ACTION aP15_FormTransporters:
(********Transporter przed dozownikami*************)
tofbFormTransportersDispencerSlow			(IN:=bFormTransportersDispencerSlowSpeedPulse, 	PT:=T#60S);
tonbFormTransportersDispencerResetSpeed		(IN:=bFormTransportersDispencerResetSpeed, 		PT:=T#5S);
tonQueBeforeScrewers						(IN:=P10_GripperScrewer.IbGripperScrewersSixthFormCheckFormSensor, PT:=T#1500mS);
tonQueAfterScrewers							(IN:=P11_CapCorrectCheck.IbCapCorrectCheckAfterScrewerFormSensor AND P11_CapCorrectCheck.IbCapCorrectCheckDialAfterScrewerFormSensor, PT:=T#2S);
tonQueAfterPlatin							(IN:=MAIN.IbLidSealerAfterSensor, PT:=T#3S);
tonQueBeforeDispencers						(IN:=MAIN.IbFormCheckFormSensor, PT:=T#2S);
tonDelayedStartAfterDisp					(IN:=NOT P09_CapPuttedCheck.fbIbCapPuttedCheckFormSensor.bOUT, PT:=T#1.5S);
IF GVL.bFormTransportersEnable AND (P00_PackML.fbPMLAuto.ePMLState = E_PMLState.ePMLState_EXECUTE)  THEN
	IF NOT VIS.bDosingTwoPhasesShow  THEN
		bFormTransportersDispencerCmdStart := TRUE;
	ELSIF VIS.bDosingTwoPhasesShow AND	NOT bFormTransportersScrewerStop AND NOT tonQueAfterPlatin.q THEN
		bFormTransportersDispencerCmdStart := TRUE;	
	END_IF
	bFormTransportersDispencerSlowSpeedPulse	:=	FALSE;
	(*Spowalnianie transportera*)	
	IF tofbFormTransportersDispencerSlow.Q AND NOT tonbFormTransportersDispencerResetSpeed.Q THEN
		bFormTransportersDispencerSlowSpeed	:= NOT VIS.bCapPuttedCheckIgnoreErrors; 
	ELSE
		bFormTransportersDispencerSlowSpeed	:= FALSE;
	END_IF
	IF bDosingTwoPhases THEN
		bFormTransportersDispencerSlowSpeed	:= TRUE;
	END_IF	
END_IF
	(*Wydmuch na tym transporterze*)
	QbBlowAfterGripperScrewer :=	bFormTransportersDispencerSlowSpeed;
(********Koniec Transporter przed dozownikami********)
	
(********Transporter za dozownikami*************)
tonbFormTransportersScrewerStop	(IN:=	(P05_Weight.eWeightStationRunningState = E_WeightLiftStationState.eStorageOfForms) AND 
										P05_Weight.fbWeightStation.iFormsCounterWeight1 >=3 AND 
										P05_Weight.fbWeightStation.iFormsCounterWeight2 >=3 AND 
										P05_Weight.fbWeightStation.iFormsCounterWeight3 >=3 AND 
										P05_Weight.fbWeightStation.iFormsCounterWeight4 >=3,
									PT:=T#500MS);
tofFormTransportersScrewerSlowSpeed	(IN:=P00_ReadRFIDCard.bReadedCardCapSorter AND bDosingTwoPhases, PT:=T#2S500MS);

IF 	P10_GripperScrewer.fbGripperScrewersDragStation.eRunningState = E_DragStationState.eEndingOfDrag  OR tonThirdFormCheckFormSensor.q THEN
//IF 	P10_GripperScrewer.fbGripperScrewersDragStation.eRunningState = E_DragStationState.eDraging AND P10_GripperScrewer.QbGripperScrewersDragLeadBefore1Actuator THEN
	bFormTransportersScrewerStop			:= FALSE;
END_IF


IF tonLongDelayAfterStart.Q AND
		eBeforeCapSorterPackageState[4].bFormPresent  AND
		(tonCapSorterFourthFormatSensorAnRegister.Q AND iCapSorterDragFormCounter >= 4)AND 
		MAIN.IbCapSorterBeforeFourthFormCheckFormSensor 
		THEN
			IF 
				NOT (
					(P05_Weight.eWeightStationRunningState = E_WeightLiftStationState.eStorageOfForms) AND 
					P05_Weight.fbWeightStation.iFormsCounterWeight1 =3 AND 
					P05_Weight.fbWeightStation.iFormsCounterWeight2 =3 AND 
					P05_Weight.fbWeightStation.iFormsCounterWeight3 =3 AND 
					P05_Weight.fbWeightStation.iFormsCounterWeight4 =3 
					)
				AND NOT bFormTransportersScrewerStop	
				//?AND NOT bLidFeederEnable
				(*AND NOT bDosingTwoPhases*)
				AND NOT bPhaseChanging
				AND tonDelayAfterStart.Q
				//AND (tonQueAfterScrewers.Q OR tonQueBeforeScrewers.Q)  //vs testy
			THEN
				bFormTransportersScrewerStop				:= 	TRUE;
			END_IF
		//bFormTransportersScrewerStop				:= 	TRUE;
END_IF
tonQueAfterScrewers.Q; tonQueBeforeScrewers.Q;
//IF bFormTransportersEnable AND (P00_PackML.fbPMLAuto.ePMLState = E_PMLState.ePMLState_EXECUTE)THEN //dp
IF bDelayAfterStart AND (*tonDelayAfterStart.Q AND*) bFormTransportersEnable AND (P00_PackML.fbPMLAuto.ePMLState = E_PMLState.ePMLState_EXECUTE OR 
		P00_PackML.fbPMLAuto.ePMLState = E_PMLState.ePMLState_STOPPING) (*AND tonDelayedStartAfterDisp.q co to*) THEN
	bFormTransportersScrewerCmdStart 			:= TRUE;
	tonbCapSorterOrCapSorterDragError.Q; 		//Spowalnianie transportera dla wag
	IF bFormTransportersScrewerStop	(*AND NOT tonbCapSorterOrCapSorterDragError.Q)*) THEN //Zatrzymywanie
		bFormTransportersScrewerCmdStart 		:= FALSE;
		
	END_IF
	//Vasyl na prośbę Karola
	(*IF (VIS.bDosingTwoPhasesShow OR vis.bLidFeederEnableShow) AND	tonQueAfterPlatin.Q OR bFormTransportersScrewerStop AND tonQueBeforeDispencers.q THEN
		bFormTransportersDispencerCmdStart 		:= FALSE;
	END_IF*)
END_IF

(********Transporter za sorterem nasadek*************)
IF bFormTransportersEnable AND (P00_PackML.fbPMLAuto.ePMLState = E_PMLState.ePMLState_EXECUTE)  THEN
	bFormTransportersAfterCapSorterCmdStart := TRUE;
	IF tonQueBeforeScrewers.Q THEN
		bFormTransportersAfterCapSorterCmdStart := FALSE;
	END_IF
END_IF	
	
(********Transporter przed zakręcarkami**************)
IF bFormTransportersEnable AND (P00_PackML.fbPMLAuto.ePMLState = E_PMLState.ePMLState_EXECUTE)  THEN
	bFormTransportersBeforeScrewerCmdStart := TRUE;
END_IF	

(*Wydmuch na tym transporterze*)
fbIbBlowBeforeGripperScrewerSensor		(bIn:=MAIN.IbBlowBeforeGripperScrewerSensor, tFilterTimeon:=T#5MS, tFilterTimeOff:=T#300MS);
fbIbBlowBeforeGripperScrewerSensor2		(bIn:=MAIN.IbBlowBeforeGripperScrewerSensor, tFilterTimeon:=T#100MS, tFilterTimeOff:=T#300MS);
tonBlowBeforeGripperScrewerSensor 		(IN:=MAIN.IbBlowBeforeGripperScrewerSensor, PT:=T#15S);
tpfbIbBlowBeforeGripperScrewerSensor 	(IN:=fbIbBlowBeforeGripperScrewerSensor.bOUT, PT:=T#1S);
QbBlowBeforeGripperScrewer	:=	fbIbBlowBeforeGripperScrewerSensor.bOut AND NOT tonBlowBeforeGripperScrewerSensor.Q;

(*Spowalniacz/szlabanik przed zakrecarkami*)
fbIbGateBeforeGripperScrewerSensor 		(bIn:=IbGateBeforeGripperScrewerSensor, tFilterTimeon:=T#20MS, tFilterTimeOff:=T#0MS);
fb2IbGateBeforeGripperScrewerSensor 	(bIn:=IbGateBeforeGripperScrewerSensor, tFilterTimeon:=T#400MS, tFilterTimeOff:=T#0MS);//bylo 670
ftfbIbGateBeforeGripperScrewerSensor	(CLK:=fbIbGateBeforeGripperScrewerSensor.bOUT,	Q=>);	
IF ftfbIbGateBeforeGripperScrewerSensor.Q THEN
	bGateBeforeGripperScrewer	:= TRUE;
END_IF
tonbGateBeforeGripperScrewer			(IN:=bGateBeforeGripperScrewer, PT:=T#400MS);
IF tonbGateBeforeGripperScrewer.Q THEN
	bGateBeforeGripperScrewer	:= FALSE;
END_IF
toniGateBeforeGripperScrewerCase1 (IN:=	iGateBeforeGripperScrewerCase = 10, PT:=T#4S);
						
CASE iGateBeforeGripperScrewerCase OF
	0:
		QbGateBeforeGripperScrewer 		:=	TRUE;
		iGateBeforeGripperScrewerCase	:=	iGateBeforeGripperScrewerCase	+	10;
	10:
		IF toniGateBeforeGripperScrewerCase1.Q AND NOT P09_CapPuttedCheck.IbCapPuttedCheckFormSensor THEN
			iGateBeforeGripperScrewerCase	:=	iGateBeforeGripperScrewerCase	+	10;
		END_IF
	20:
		QbGateBeforeGripperScrewer		:=	FALSE;
		iGateBeforeGripperScrewerCase	:=	iGateBeforeGripperScrewerCase	+	10;
	30: 
		QbGateBeforeGripperScrewer :=		fb2IbGateBeforeGripperScrewerSensor.bOUt;
END_CASE
	
//Spowalnianie formatek
iFormBeforeScrewers := 		
                       		BOOL_TO_INT(eBeforeScrewers2PackageState[2].bFormPresent)+
                       		BOOL_TO_INT(eBeforeScrewers2PackageState[1].bFormPresent)+
                       		BOOL_TO_INT(eBeforeScrewersPackageState[2].bFormPresent)+
                       		BOOL_TO_INT(eBeforeScrewersPackageState[1].bFormPresent);

tonCapPuttedFormsCheck			(IN:=	P10_GripperScrewer.IbGripperScrewersSixthFormCheckFormSensor,		PT:=T#80MS); //bylo 130
tonThirdFormCheckFormSensor		(IN:=	NOT P10_GripperScrewer.IbGripperScrewersSixthFormCheckFormSensor ,	PT:=T#30MS);
IF // Zatrzymywanie jeżeli
	tonCapPuttedFormsCheck.Q OR 			
	P00_PackML.fbPMLAuto.ePMLState = E_PMLState.ePMLState_STOPPING 	OR	
	NOT tonDelayAfterStart.Q	
THEN
	bFormTransporterSlowerCmdStart := FALSE;
END_IF
IF bDelayAfterStart AND bFormTransportersEnable AND 
	(
		tonThirdFormCheckFormSensor.Q OR 
		(NOT bDelayAfterStartFullRegister AND NOT P09_CapPuttedCheck.IbCapPuttedCheckFormSensor) OR
		(bDelayAfterStartFullRegister AND iFormBeforeScrewers=2) //do usuniecia
	)
	AND
	NOT (P00_PackML.fbPMLAuto.ePMLState = E_PMLState.ePMLState_STOPPING) 
	THEN 
		bFormTransporterSlowerCmdStart := TRUE;
END_IF

(********Transporter za zakręcarkami**************)
IF bFormTransportersEnable AND (P00_PackML.fbPMLAuto.ePMLState = E_PMLState.ePMLState_EXECUTE)  THEN
	bFormTransportersAfterScrewerCmdStart := TRUE;
END_IF
END_ACTION

ACTION aP16_LabelMachines:
(***********P16_LabelMachines**************)
(******************************************)
IF bLabelMachineEnable THEN
	bLabelMachineCmdStart := TRUE;
ELSE
	bLabelMachineCmdStart := FALSE;	
END_IF
(******************************************)
(******************************************)
END_ACTION

ACTION aP17_TurnTables:
(************P17_TurnTables****************)
(******************************************)

IF bExitTurnTableEnable AND bDelayAfterStart THEN
	bExitTurnTableCmdStart := TRUE;
ELSIF bDelayAfterStart THEN
	;//bExitTurnTableCmdStart := FALSE;
END_IF
(******************************************)
(******************************************)
IF bExitConveyorEnable AND bDelayAfterStart THEN
	bExitConveyorCmdStart := TRUE;
ELSE
	;//bExitConveyorCmdStart := FALSE;
END_IF
(******************************************)
(******************************************)


(*********************************************************)
(*********Szlaban na transporterze odbiorczym*************)
//Jeżeli stół pracuje 
bExitConveyorCmdStart;
//To ruszaj szlabanem
bExitConveyorGateRun;
//Czujnik z szlabanem
P17_TurnTables.IbExitConveyorGateAfterSensor;
P17_TurnTables.IbExitConveyorGateAfterSensor2;
IF bExitConveyorCmdStart THEN
	fbIbExitConveyorGateAfterSensor		(bIN:=P17_TurnTables.IbExitConveyorGateAfterSensor,	tFilterTimeOn:=T#10MS,	tFilterTimeOff:=T#10MS);
	fbIbExitConveyorGateAfterSensor2	(bIN:=P17_TurnTables.IbExitConveyorGateAfterSensor2,tFilterTimeOn:=T#1S800MS,	tFilterTimeOff:=T#1S800MS);
	tonbExitConveyorGateRun				(IN:=bExitConveyorGateRun AND NOT fbIbExitConveyorGateAfterSensor.bOUT, 	PT:=T#300MS);
	
	bExitConveyorGateRun S= fbIbExitConveyorGateAfterSensor.bOut;	
	bExitConveyorGateRun R= tonbExitConveyorGateRun.Q;	
	
	IF fbIbExitConveyorGateAfterSensor2.bOut AND bExitConveyorGateRun THEN
		bExitConveyorGateRunTemp := TRUE;
	ELSIF NOT fbIbExitConveyorGateAfterSensor2.bOut THEN
		bExitConveyorGateRunTemp := FALSE;	
	END_IF
	IF bExitConveyorGateRunTemp THEN
		bExitConveyorGateRun	:=	TRUE;
	END_IF
END_IF
(*********************************************************)
(*********************************************************)
	fbIbExitConveyorGateAfterSensor3		(bIN:=P17_TurnTables.IbExitConveyorGateAfterSensor,	tFilterTimeOn:=T#10MS,	tFilterTimeOff:=T#12S);

IF tonNotExecute.Q AND NOT fbIbExitConveyorGateAfterSensor3.bOut THEN
	bExitTurnTableCmdStart := FALSE;
	bExitConveyorCmdStart := FALSE;
END_IF
END_ACTION

END_PROGRAM

// ---- POUs/P00_Visualization.TcPOU
PROGRAM P00_Visualization
VAR
	iCaseDialogResetCycle				: INT;
	iCaseDialogHoming					: INT;
	iCaseDialogOpenDoors				: INT;
	iCaseDialogWeighing					: INT;
	iCaseDialog2Phase					: INT;
	iCaseDialogExMode					: INT;
	
	tonTimerCycleReseting				: TON;
	bCycleResetDone						: BOOL;
	(*Informacyjne*)

	
	tonCaseDialogHomingCase30: TON;
	tonCaseDialogGomingResetting: TON;
	rtChangeOver: R_TRIG;
	ftChangeOver: F_TRIG;
	iEmergencyOpen: INT;
	tonEStopDoorsDelayOpen: TON;
	rtbDosingTwoPhasesShow: R_TRIG;
	ftbDosingTwoPhasesShow: F_TRIG;
	ftbExModeOn: F_TRIG;
	rtbExModeOn: R_TRIG;
	rtIbSafetyResetIn		:	R_TRIG;
	tonCycleStopButton		:	TON;
	rtIbEmergencyStopButton	:	R_TRIG;
	bEStopButtonPressed	:	BOOL;
		
	(*Wyświetlanie informacji*)
	//fbInformationDisplay				: FB_InformationDisplay;
	AbInformationOnTemp					: ARRAY[0..63] OF BOOL;	// Tablica informacji	
	AudiInformationDescriptionIDTemp	: ARRAY[0..63] OF UDINT;

	n									: INT;
	(*Inne*)
	
	tonNoFormsBeforeDispencers: TON;
	fbTcTouchLock_AcquireFocus: FB_TcTouchLock_AcquireFocus;
	bSORNHoming: BOOL;
	temp: BOOL;
	
	pvStationInError: PVOID;
	
	temp2: BOOL;
	tonStringtoWstring: TON;
	bStringtoWstring1: BOOL;
	bStringtoWstring2: BOOL;
	bStringtoWstring3: BOOL;
	bStringtoWstring4: BOOL;
	rtbStringtoWstring1: R_TRIG;
	rtbStringtoWstring2: R_TRIG;
	rtbStringtoWstring3: R_TRIG;
	rtbStringtoWstring4: R_TRIG;
	rtInformationNew: R_TRIG;
	iAbInformationOnTempCounterTemp: INT;
	tonInformationNew: TON;
	sWeightTime: STRING;
	tonInformation: TON;
	rtStartAck :R_TRIG;
	ftStopCancel: F_TRIG;
	tonbDialogBoxAckAndCancel:TON;
END_VAR

aStringToWString();
ACT_MachineStatus();
ACT_DoorsUnlock();
ACT_Homing();
ACT_Info();
//ACT_Weighting();

Information();
aEstopDoors();
aTouchScreen();
aBottleDelete();
aStartStopButtons();

ACTION aBottleDelete:
IF 	VIS.bBottleDeleteUnderDispencers	THEN
	
	 eBeforeDispencersPackageState[4].bBottlePresent		:=	FALSE;	
	 eBeforeDispencersPackageState[3].bBottlePresent		:=	FALSE;
	 eBeforeDispencersPackageState[2].bBottlePresent		:=	FALSE;
	 eBeforeDispencersPackageState[1].bBottlePresent		:=	FALSE;
	
	
	 eDispencersPackageState[4].bBottlePresent				:=	FALSE; 
	 eDispencersPackageState[3].bBottlePresent				:=	FALSE;
	 eDispencersPackageState[2].bBottlePresent				:=	FALSE; 
	 eDispencersPackageState[1].bBottlePresent				:=	FALSE; 
	
	 eBeforeDispencer12PackageState2Phase[2].bBottlePresent	:=	FALSE;
	 eBeforeDispencer12PackageState2Phase[1].bBottlePresent	:=	FALSE; 
	 
	 eBeforeDispencer34PackageState2Phase[2].bBottlePresent	:=	FALSE;
	 eBeforeDispencer34PackageState2Phase[1].bBottlePresent	:=	FALSE;
	 
	 eDispencer12PackageState2Phase[2].bBottlePresent		:=	FALSE;
	 eDispencer12PackageState2Phase[1].bBottlePresent		:=	FALSE;
	 
	 eDispencer34PackageState2Phase[2].bBottlePresent		:=	FALSE;
	 eDispencer34PackageState2Phase[1].bBottlePresent		:=	FALSE;
	 
	 VIS.bBottleDeleteUnderDispencers	:=	FALSE;
	 
END_IF
END_ACTION

ACTION ACT_DoorsUnlock:

(*** DO PRZETESTOWANIA**)

(****** Komunikat pytania 'Czy odblokować drzwi *****)

CASE iCaseDialogOpenDoors OF
	
	0:
		IF VIS.bDoorsUnlock THEN
			iCaseDialogOpenDoors:= 1;
		END_IF
			
	1: 
		IF 	 QbDispencersDoorsClose AND QbLidSealingDoorsClose AND QbGripperScrewerClose AND QbBottleTransferDoorsClose AND QbTanksDoorsClose AND QbPickInserterDoorsClose AND P07_ROPP.QbROPPDoors0Close AND P07_ROPP.QbROPPDoors1Close	THEN
			iCaseDialogOpenDoors:= 2;
		ELSE
			iCaseDialogOpenDoors:= 3;	
		END_IF
		
	2:
		VIS.nDialogBoxType		:= 3;	// Rodzaj okna, 0-nic, 1-tylko przysisk OK, 2 - tylko przycisk Anuluj, 3 - Przycisk OK i Anuluj
		VIS.bDialogBoxText		:= 'Unlock the doors?';
		VIS.sDialogBoxPicture	:= 'info';
		VIS.bDialogBoxOn		:= TRUE;
		IF VIS.bDialogBoxAck THEN
			VIS.bDialogBoxAck			:=	FALSE;				// Zawsze kasuj OK po naciśnięciu
			iCaseDialogOpenDoors:= 4;
		ELSIF VIS.bDialogBoxCancelAck THEN	
			VIS.bDialogBoxCancelAck		:=FALSE; 
			iCaseDialogOpenDoors:= 5;
		END_IF
		
	3:
		
		QbDispencersDoorsClose		  	:= TRUE;
		QbLidSealingDoorsClose			:= TRUE;	
		QbGripperScrewerClose		   	:= TRUE;	
		QbBottleTransferDoorsClose		:= TRUE;	
		QbTanksDoorsClose				:= TRUE;
		QbPickInserterDoorsClose		:= TRUE;
		VIS.nDialogBoxType				:=	1;										// Rodzaj okna, 0-nic, 1-tylko przysisk OK, 2 - tylko przycisk Anuluj, 3 - Przycisk OK i Anuluj
		VIS.bDialogBoxText				:=	'Doors loked';
		VIS.sDialogBoxPicture			:= 'info';
		VIS.bDialogBoxOn				:=	TRUE;	
	
		IF VIS.bDialogBoxAck THEN
			iCaseDialogOpenDoors:= 5;	
			VIS.bDialogBoxAck				:=	FALSE;				// Zawsze kasuj OK po naciśnięciu	
		END_IF
		
	4:
		QbDispencersDoorsClose		  	:= FALSE;	
		QbLidSealingDoorsClose			:= FALSE;
		QbGripperScrewerClose		   	:= FALSE;	
		QbBottleTransferDoorsClose		:= FALSE;
		QbTanksDoorsClose				:= FALSE;
		QbPickInserterDoorsClose		:= FALSE;
		VIS.nDialogBoxType				:=	1;					// Bez przycisków
		VIS.bDialogBoxText				:=	'Doors unlocked';	
		VIS.sDialogBoxPicture			:= 'uwaga';
		IF VIS.bDialogBoxAck THEN
			iCaseDialogOpenDoors:= 5;		
		END_IF
	
	5:
		VIS.bDoorsUnlock 		:= FALSE;								
		aResetDialog();
		iCaseDialogOpenDoors	:= 0;
		
END_CASE

//Dodane otwieranie drzwi przy przyzbrajaniu LU205
rtChangeOver(CLK:=bChangeOver,Q=>);
ftChangeOver(CLK:=bChangeOver,Q=>);
(*IF rtChangeOver.Q THEN
		QbDispencersDoorsClose		   		:= FALSE;	
		QbGripperScrewerClose		   		:= FALSE;	
		QbBottleTransferDoorsClose			:= FALSE;	
END_IF
IF ftChangeOver.Q THEN
		QbDispencersDoorsClose		   		:= FALSE;	
		QbGripperScrewerClose		    	:= FALSE;	
		QbBottleTransferDoorsClose			:= FALSE;	
END_IF*)
END_ACTION

ACTION ACT_Homing:


tonCaseDialogHomingCase30(IN := iCaseDialogHoming = 30, PT := T#3S);
tonCaseDialogGomingResetting(IN := P00_PackML.fbPMLAuto.ePMLState = E_PMLState.ePMLState_RESETTING, PT := T#2S);

(****** Komunikat pytania 'Czy bazować" *****)
CASE iCaseDialogHoming OF
    0:
        IF tonCaseDialogGomingResetting.Q THEN
            IF bHomingDialog THEN
                iCaseDialogHoming := 10;
            END_IF
        END_IF

	10:	
        VIS.nDialogBoxType    := 3; // Rodzaj okna, 0-nic, 1-tylko przycisk OK, 2 - tylko przycisk Anuluj, 3 - Przycisk OK i Anuluj
        VIS.bDialogBoxText    := 'Start homing?';
        VIS.sDialogBoxPicture := 'info';
        VIS.bDialogBoxOn      := TRUE;
        VIS.sDialogBoxPicture := '';
		
		IF NOT P00_PackML.bStationsAreReadyOrManual THEN
			VIS.bDialogBoxText2    := Concat('Stations are not ready, wait ',sHomingText);
			VIS.bDialogBoxAck		:= FALSE;
		ELSE
			VIS.bDialogBoxText2    := Concat('Stations ready ',sHomingText);
			IF NOT (sHomingText = '') THEN
				VIS.bDialogBoxText2    := Concat('Stations ready, homing of the stations: ',sHomingText);
			END_IF
		END_IF		
		
		VIS.bDialogBoxAckNeeded			:= TRUE;
        IF VIS.bDialogBoxAck THEN
			VIS.bDialogBoxAck 			:= FALSE;
			VIS.bDialogBoxAckNeeded		:= FALSE;
			
			//IF bRecipeChangePositioning THEN
			//	bCycleReseting := TRUE;	 NIE DZIAŁA
			//END_IF
			
            iCaseDialogHoming 			:= iCaseDialogHoming + 10;
			
			// Dodatkowy komunikat
			IF sHomingText = 'SORN,' THEN
				bSORNHoming	:=	TRUE;
			END_IF
			
			
        ELSIF VIS.bDialogBoxCancelAck THEN
			bHomingCanceled				:= TRUE;
			bRecipeChangePositioning 	:= FALSE;
			VIS.bDialogBoxAckNeeded		:= FALSE;
            iCaseDialogHoming := 30;//20;
        END_IF

    20:
        VIS.bDialogBoxAck     := FALSE; // Zawsze kasuj OK po naciśnięciu
        VIS.nDialogBoxType    := 0;     // Bez przycisków
        VIS.bDialogBoxText    := 'Homing ... ';
        VIS.bDialogBoxText2   := sHomingText;
        VIS.sDialogBoxPicture := '';
        bHoming               := TRUE;

		IF bRecipeChangePositioning THEN //Kasowanie korekt tylko dla wybrania całej nowej receptury
			
			VIS.bBadPackageReasonReset := TRUE;
			VIS.uiCounterAverageEfficiency:=0;
			VIS.udiCounterShiftBottles:=0;
			VIS.uiCounterInstantEfficiency:=0;
			VIS.uiCounterGoodBottles:=0;
			VIS.uiCounterBadBottles:=0;
			VIS.udiCounterGlobalBadBottles:=0;
			VIS.bOEEGenRaport	:=	TRUE;
		END_IF

    	 iCaseDialogHoming := iCaseDialogHoming + 10;
	30:	
		(*Jeżeli bazownia zostały wyłączone*)
        IF tonCaseDialogHomingCase30.Q AND NOT P00_PackML.bHomingIsOnAtLeastOneStation THEN
            iCaseDialogHoming := iCaseDialogHoming + 10;
        END_IF

    40:
	
		IF bHomingCanceled THEN
			VIS.nDialogBoxType    	:= 1;
			VIS.bDialogBoxText    	:= 'Homing canceled';
			VIS.sDialogBoxPicture 	:= '1';
			VIS.bDialogBoxOn      	:= TRUE;
			VIS.bDialogBoxAckNeeded	:= TRUE;
		ELSE
			VIS.nDialogBoxType    	:= 1;
			VIS.bDialogBoxText    	:= 'Homing done';
			IF bSORNHoming THEN
				VIS.bDialogBoxText    	:= 'Clean up the closings after the homing';	
			END_IF
			VIS.sDialogBoxPicture 	:= '1';
			VIS.bDialogBoxOn      	:= TRUE;
			VIS.bDialogBoxAckNeeded	:= TRUE;			
		END_IF
        IF VIS.bDialogBoxAck THEN
			bSORNHoming				:= FALSE;
			VIS.bDialogBoxAck		:= FALSE;
			VIS.bDialogBoxAckNeeded	:= FALSE;
            iCaseDialogHoming 		:= iCaseDialogHoming + 10;
        END_IF

    50:
        bHomingDialog := FALSE;
        aResetDialog();
        iCaseDialogHoming := 0;

END_CASE

(****** Koniec Komunikat pytania 'Czy resetować" *****)
END_ACTION

ACTION ACT_Info:
(****** Komunikat pytania 'Czy resetować" *****)

CASE iCaseDialogResetCycle OF
	
	0:
		IF P00_PackML.fbPMLModeManager.eModeStatus = E_PMLUnitMode.ePMLUnitMode_AUTOMATIC AND P00_PackML.fbPMLAuto.ePMLState = E_PMLState.ePMLState_IDLE THEN
			IF VIS.bCycleReset  THEN
				iCaseDialogResetCycle:= 1;
			END_IF
		END_IF	
		
	1:
		VIS.nDialogBoxType		:= 3;													// Rodzaj okna, 0-nic, 1-tylko przysisk OK, 2 - tylko przycisk Anuluj, 3 - Przycisk OK i Anuluj
		VIS.bDialogBoxText		:= 'Perform cycle reset?';
		VIS.sDialogBoxPicture	:= 'info';
		VIS.bDialogBoxOn		:= TRUE;
		VIS.sDialogBoxPicture	:= '';
	
		IF VIS.bDialogBoxAck THEN
			VIS.bDialogBoxAck := FALSE;
			iCaseDialogResetCycle:= 2;
		ELSIF VIS.bDialogBoxCancelAck THEN	
			iCaseDialogResetCycle:= 3;
		END_IF

	2:
		bCycleReseting			:= TRUE;											// Jeżeli OK to zacznij
		VIS.bDialogBoxAck		:= FALSE;											// Zawsze kasuj OK po naciśnięciu
		VIS.nDialogBoxType		:= 0;												// Bez przycisków
		VIS.bDialogBoxText		:= 'Cycle reset...';	
		VIS.sDialogBoxPicture	:= '';
		
		IF tonTimerCycleReseting.Q THEN // po 2 sekundach
			iCaseDialogResetCycle:= 4;
		END_IF

	3:	
		bCycleReseting			:= FALSE;
		VIS.bCycleReset			:= FALSE;								
		aResetDialog();
		iCaseDialogResetCycle:= 0;

	4:
		bCycleReseting			:= FALSE;								
		VIS.nDialogBoxType		:= 1;
		VIS.bDialogBoxText		:= 'Cycle reset done';
		VIS.sDialogBoxPicture	:= '1';
		VIS.bDialogBoxOn		:= TRUE;
		bCycleResetDone 		:= TRUE;
		IF bCycleResetDone AND VIS.bDialogBoxAck THEN
			VIS.bDialogBoxAck := FALSE;
			iCaseDialogResetCycle:= 5;
		END_IF

	5:
		bCycleResetDone 		:= FALSE;
		VIS.bCycleReset			:= FALSE;								
		aResetDialog();
		iCaseDialogResetCycle:= 0;

END_CASE

(****** Koniec Komunikat pytania 'Czy resetować" *****)



tonTimerCycleReseting.IN 			:= iCaseDialogResetCycle = 2;
tonTimerCycleReseting.PT 			:= T#2S;
tonTimerCycleReseting();
END_ACTION

ACTION ACT_MachineStatus:

(** Przygotowanie zmiennych dla Wizki*)
VIS.iMachineState	:=		INT_TO_UINT(P00_PackML.fbPMLAuto.ePMLState);

CASE P00_PackML.fbPMLAuto.ePMLState OF
	
	E_PMLState.ePMLState_ABORTING:
		VIS.sMachineState				:= 'ABORTING' ;
		
	E_PMLState.ePMLState_ABORTED:
		VIS.sMachineState				:= 'ABORTED' ;		
		
	E_PMLState.ePMLState_STOPPING:
		VIS.sMachineState				:= 'STOPPING' ;
		
	E_PMLState.ePMLState_STOPPED:	
		VIS.sMachineState				:= 'STOPPED,ERROR' ;	
	
	E_PMLState.ePMLState_RESETTING:
		VIS.sMachineState				:= 'RESETTING' ;
	
	E_PMLState.ePMLState_IDLE:	
		VIS.sMachineState				:= 'IDLE' ;
		
	E_PMLState.ePMLState_STARTING:
		VIS.sMachineState				:= 'STARTING' ;
			
	E_PMLState.ePMLState_EXECUTE:
		VIS.sMachineState				:= 'EXECUTE' ;
			
	E_PMLState.ePMLState_COMPLETING:
		VIS.sMachineState				:= 'COMPLETING';
		
	E_PMLState.ePMLState_COMPLETE:
		VIS.sMachineState				:= 'COMPLETE';
		
	E_PMLState.ePMLState_UNDEFINED:
		VIS.sMachineState				:= 'UNDEFINED';
		
END_CASE


IF P00_PackML.fbPMLModeManager.eModeStatus = E_PMLUnitMode.ePMLUnitMode_MANUAL THEN
	VIS.sMachineState	:=	CONCAT('MANUAL MODE | ',VIS.sMachineState);
END_IF

IF P00_PackML.fbPMLModeManager.eModeStatus = E_PMLUnitMode.ePMLUnitMode_AUTOMATIC THEN
	VIS.sMachineState	:=	CONCAT('AUTO | ',VIS.sMachineState);
END_IF

IF P00_PackML.fbPMLModeManager.eModeStatus = E_PMLUnitMode.ePMLUnitMode_UNDEFINED THEN
	VIS.sMachineState	:=	CONCAT('NIEZNANY | ',VIS.sMachineState);
END_IF
END_ACTION

ACTION ACT_Weighting:
(****** Komunikat pytania 'Czy wykonać przeważenie formatek *****)


CASE iCaseDialogWeighing OF
	
	0:
	
		IF P00_PackML.fbPMLModeManager.eModeStatus = E_PMLUnitMode.ePMLUnitMode_AUTOMATIC AND P00_PackML.fbPMLAuto.ePMLState = E_PMLState.ePMLState_STARTING THEN
		
			IF NOT MAIN.bWeighingFormDone THEN
				iCaseDialogWeighing				:= 10;
			END_IF
	
		END_IF
	
	10:
	
		VIS.nDialogBoxType						:= 3;
		VIS.bDialogBoxText						:= 'Perform reweighing pucks  ?';
		VIS.sDialogBoxPicture					:= 'info';
		VIS.bDialogBoxOn						:= TRUE;
		VIS.sDialogBoxPicture					:= '';
		
		IF VIS.bDialogBoxAck THEN
			iCaseDialogWeighing					:= 20;
		END_IF
	
		IF VIS.bDialogBoxCancelAck THEN
			iCaseDialogWeighing					:= 30;
		END_IF
		
	20:
	
		VIS.bWeighingForm						:= TRUE;
		iCaseDialogWeighing						:= 30;
		
	30:
	
		aResetDialog();
		iCaseDialogWeighing						:= 0;
				
END_CASE
END_ACTION

ACTION aEstopDoors:
/// Automatyczne odryglowanie drzwi po wciśnietym grzybie

(* Po wcisnieciu grzyba czeka 2 sekundy, a potem odryglowuje wszystkie drzwi*)
(* Trzeba dwa razy wciskać przycisk resetu *)
(* Pierwszy reset resetuje grzyby, a drugi rygle*)
//tonCycleStopButton (IN:=NOT IbCycleStopButton AND QbDispencersDoorsClose , PT:=T#3S);

tonCycleStopButton (IN:=	(
//							NOT	IbCycleStopButton OR NOT IbTurnTableCycleStopButton OR NOT P07_ROPP.IbROPPCycleStopButton OR
							NOT	IbCycleStopButton  (*OR NOT P07_ROPP.IbROPPCycleStopButton OR	NOT IbPucksInserterCycleStopButton*)	OR	
							(NOT stBottleSorterRead.bCycleStop	AND NOT bBottleSorterDisable) OR 
							(NOT stCapSorterRead.bCycleStop		AND NOT bCapSorterDisable)
							)
							AND QbDispencersDoorsClose , PT:=T#1S500MS);



//rtIbSafetyResetIn	(CLK:=IbSafetyResetIn,  Q=>);
rtIbSafetyResetIn	(CLK:=IbSafetyResetIn OR QbSafetyResetBottleSorterIn OR QbSafetyResetCapSorterIn,  Q=>);
IF rtIbSafetyResetIn.Q  THEN
	QbDispencersDoorsClose		   		:= TRUE;	
	QbLidSealingDoorsClose				:= TRUE;
	QbGripperScrewerClose		    	:= TRUE;	
	QbBottleTransferDoorsClose			:= TRUE;
	QbTanksDoorsClose					:= TRUE;
	QbPickInserterDoorsClose			:= TRUE;
END_IF

rtIbEmergencyStopButton	(CLK:=bEStopButtonPressed OR tonCycleStopButton.Q, Q=>);
IF rtIbEmergencyStopButton.Q THEN
	QbDispencersDoorsClose		   		:= FALSE;
	QbLidSealingDoorsClose				:= FALSE;
	QbGripperScrewerClose		    	:= FALSE;	
	QbBottleTransferDoorsClose			:= FALSE;
	QbTanksDoorsClose					:= FALSE;
	QbPickInserterDoorsClose			:= FALSE;
	
END_IF


bEStopButtonPressed := IbEmergencyStopButton0Pressed OR IbEmergencyStopButton1Pressed OR IbEmergencyStopButton2Pressed OR IbEmergencyStopButton3Pressed OR IbEmergencyStopButton4Pressed OR 
						IbTurnTableEmergencyStopButtonPressed OR 
						IbPucksInserterEmergencyStopButton0Pressed OR IbPucksInserterEmergencyStopButton1Pressed OR 
						P07_ROPP.IbROPPEmergencyStopButton0Pressed OR P07_ROPP.IbROPPEmergencyStopButton1Pressed OR 
						bCapSorterEmergencyStopButton1Pressed OR bCapSorterEmergencyStopButton2Pressed OR bCapSorterEmergencyStopButton3Pressed;

tonEStopDoorsDelayOpen(IN:=iEmergencyOpen=10, PT:=T#2000MS);
(*
CASE iEmergencyOpen OF


		0:
			IF bEStopButtonPressed THEN
			//IF NOT GVL_IO.IbEmergencyStopButton THEN
				iEmergencyOpen:=10;
			END_IF
			
		10:
			//Otwarcie drzwi - podanie zasilania na cewki rygli
			IF tonEStopDoorsDelayOpen.Q THEN
				QbDispencersDoorsClose		   		:= FALSE;	
				QbGripperScrewerClose		    	:= FALSE;		
				QbBottleTransferDoorsClose			:= FALSE;	
			END_IF;
			
			//IF GVL_IO.IbEmergencyStopButton THEN			
			IF bEStopButtonPressed THEN
				iEmergencyOpen:=20;
			END_IF
		20:
			//zamknięci drzwi - zaryglowanie
			QbDispencersDoorsClose		   		:= TRUE;
			QbGripperScrewerClose		    	:= TRUE;
			QbBottleTransferDoorsClose			:= TRUE;
			iEmergencyOpen:=0;
		
	
END_CASE
*)
END_ACTION

ACTION aResetDialog:
VIS.nDialogBoxType	:=	0;
VIS.bDialogBoxText	:=	'';
VIS.bDialogBoxText2	:=	'';
VIS.sDialogBoxPicture	:= '';
VIS.bDialogBoxOn	:=	FALSE;
VIS.bDialogBoxCancelAck	:=	FALSE;
VIS.bDialogBoxAck	:=	FALSE;
END_ACTION

ACTION aStartStopButtons:
rtStartAck														(CLK:= (IbCycleStartButton OR IbTurnTableCycleStartButton OR P07_ROPP.IbROPPCycleStartButton OR IbPucksInserterCycleStartButton OR
																		(stBottleSorterRead.bCycleStart AND NOT bBottleSorterDisable) OR
																		(stCapSorterRead.bCycleStart AND NOT bCapSorterDisable)) );
																
ftStopCancel													(CLK:= 	NOT		IbCycleStopButton OR NOT IbTurnTableCycleStopButton OR NOT P07_ROPP.IbROPPCycleStopButton OR NOT IbPucksInserterCycleStopButton OR
																		(NOT	stBottleSorterRead.bCycleStop	AND NOT bBottleSorterDisable) OR 
																		(NOT	stCapSorterRead.bCycleStop		AND NOT bCapSorterDisable) );
																		

IF rtStartAck.Q THEN
	VIS.bDialogBoxAck 			:= TRUE;
END_IF
IF ftStopCancel.Q THEN
	VIS.bDialogBoxCancelAck 	:= TRUE;
END_IF


tonbDialogBoxAckAndCancel (IN:=VIS.bDialogBoxAck OR VIS.bDialogBoxCancelAck, PT:=T#1S);
IF tonbDialogBoxAckAndCancel.Q THEN
	VIS.bDialogBoxAck 			:= FALSE;
	VIS.bDialogBoxCancelAck		:= FALSE;	
END_IF
END_ACTION

ACTION aStringToWString:
//VIS.wsStationInError			:=	"polskie znaki ąśźżłóćęŁĄĆŚŻŹ¹";
									//	STRING_TO_WSTRING(VIS.sStationInError);
//VIS.wsStationErrorDescription	:=	STRING_TO_WSTRING(VIS.sStationErrorDescription);

//VIS.wsStationErrorDescription	:=	UTF8_TO_WSTRING(STRING_TO_UTF8(VIS.sStationErrorDescription));	
//VIS.wsStationErrorDescription2	:=	STRING_TO_WSTRING(VIS.sStationErrorDescription2);
//VIS.sStationInError:=wsLiteral_TO_UTF8(VIS.sStationInError);

//temp:=STRING_TO_UTF8	(pDstUTF8:=pvStationInError, pSrcSTRING:=ADR(VIS.sStationInError), nDstSize:=SIZEOF(VIS.sStationInError));
//temp2:=UTF8_TO_WSTRING	(pDstWSTRING:= ADR(VIS.wsStationInError), pSrcUTF8:=pvStationInError , nDstSize:=SIZEOF(VIS.wsStationInError), nDstLen=> );


//temp:=STRING_TO_WSTRING2(pDstWSTRING:=ADR(VIS.wsStationInError), pSrcSTRING:=ADR(VIS.sStationInError), nDstSize:=SIZEOF(VIS.wsStationInError));

tonStringtoWstring(IN:=NOT tonStringtoWstring.Q, PT:=T#1200MS);
IF tonStringtoWstring.ET > T#10MS AND NOT tonStringtoWstring.Q THEN
	bStringtoWstring1	:=	TRUE;
END_IF
IF tonStringtoWstring.ET > T#300MS AND NOT tonStringtoWstring.Q THEN
	bStringtoWstring2	:=	TRUE;
END_IF
IF tonStringtoWstring.ET > T#600MS AND NOT tonStringtoWstring.Q THEN
	bStringtoWstring3	:=	TRUE;
END_IF
IF tonStringtoWstring.ET > T#900MS AND NOT tonStringtoWstring.Q THEN
	bStringtoWstring4	:=	TRUE;
END_IF
IF tonStringtoWstring.Q THEN
	bStringtoWstring1	:=	bStringtoWstring2	:=	bStringtoWstring3	:=	bStringtoWstring4	:= FALSE;
END_IF
rtbStringtoWstring1	(CLK:=bStringtoWstring1, Q=>);
rtbStringtoWstring2	(CLK:=bStringtoWstring2, Q=>);
rtbStringtoWstring3	(CLK:=bStringtoWstring3, Q=>);
rtbStringtoWstring4	(CLK:=bStringtoWstring4, Q=>);

IF rtbStringtoWstring1.Q THEN
	VIS.wsStationInError			:=	F_StringToWstringPL(sInput:=VIS.sStationInError);
	VIS.wsStationErrorDescription	:=	F_StringToWstringPL(sInput:=VIS.sStationErrorDescription);
	VIS.wsStationErrorDescription2	:=	F_StringToWstringPL(sInput:=VIS.sStationErrorDescription2);	
	VIS.wsMachineState				:=	F_StringToWstringPL(sInput:=VIS.sMachineState);
END_IF
	
IF rtbStringtoWstring2.Q THEN	
	VIS.wsDialogBoxText				:=	F_StringToWstringPL(sInput:=VIS.bDialogBoxText);
	VIS.wsDialogBoxText2			:=	F_StringToWstringPL(sInput:=VIS.bDialogBoxText2);
	VIS.wsBadPackageReason1			:=	F_StringToWstringPL(sInput:=VIS.sBadPackageReason1);
	VIS.wsBadPackageReason2			:=	F_StringToWstringPL(sInput:=VIS.sBadPackageReason2);
	VIS.wsBadPackageReason3			:=	F_StringToWstringPL(sInput:=VIS.sBadPackageReason3);
END_IF
	
IF rtbStringtoWstring3.Q THEN				
	VIS.wsSlowestStation1			:=	F_StringToWstringPL(sInput:=VIS.sSlowestStation1);	
	VIS.wsSlowestStation2			:=	F_StringToWstringPL(sInput:=VIS.sSlowestStation2);	
	VIS.wsSlowestStation3			:=	F_StringToWstringPL(sInput:=VIS.sSlowestStation3);	
	VIS.wsSlowestStation4			:=	F_StringToWstringPL(sInput:=VIS.sSlowestStation4);	
END_IF
	
IF rtbStringtoWstring4.Q THEN
	VIS.wsSlowestStation5			:=	F_StringToWstringPL(sInput:=VIS.sSlowestStation5);	
	//bylo 	AsActiveWarningDescription				:ARRAY [0..63] OF STRING;	//  Aktywne ostrzeżenia
	//jest	AwsActiveWarningDescription				:ARRAY [0..63] OF WSTRING;	//  Aktywne ostrzeżenia
	//FOR i := 0 TO 63-1 DO
	//	VIS.AwsInformationDescription[i] :=	F_StringToWstringPL(sInput:=VIS.AsInformationDescription[i]);
	//END_FOR
END_IF
END_ACTION

ACTION aTouchScreen:
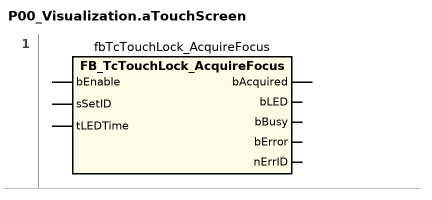
// NETWORK 1
fbTcTouchLock_AcquireFocus(); // FB_TcTouchLock_AcquireFocus
END_ACTION

ACTION Information:
(*
Nazwa:			Information
Wersja:			v0.1 			
Autor:			DP
Urzadzenia:		HMI, 
Konfiguracja:	
	AsInformationDescription  	: ARRAY[0..63] OF STRING; // Opis informacji, tablica na stałe wypisana
Info:
- Segregacja tekstów od tablicy 0,
- Wizualizacja wyświetla Informację tj.: Koniec konfekcji,
Uwagi:

Zmiany:

*)

VIS.AsInformationDescription[0];
VIS.AsInformationDescription[1];

tonNoFormsBeforeDispencers(	IN:= NOT MAIN.IbFormCheckFormSensor AND NOT MAIN.IbFourthFormCheckFormSensor  AND (P00_PackML.fbPMLAuto.ePMLState = E_PMLState.ePMLState_EXECUTE), PT:= T#20S);
tonInformation			  (IN:= NOT tonInformation.Q,	PT:=T#1S);

//IF tonInformation.Q THEN
	(**KROK 1**)
	(**Czyszczenie tablicy**)
	FOR i := 0 TO 63-1 DO
		VIS.AsInformationDescription[i] := '';
		VIS.AStInformationDescription[i].udiID := 0;
		VIS.AStInformationDescription[i].wsDescription := "";	
	END_FOR
	
	(**KROK 2**)
	(**Wpisywanie komunikatów**)
	AbInformationOnTemp[0]								:=	NOT QbDispencersDoorsClose OR  NOT QbLidSealingDoorsClose OR NOT QbGripperScrewerClose OR NOT QbBottleTransferDoorsClose OR NOT QbTanksDoorsClose OR NOT QbPickInserterDoorsClose OR NOT P07_ROPP.QbROPPDoors0Close	OR NOT P07_ROPP.QbROPPDoors0Close;
	VIS.AsInformationDescription[0]						:=	'Drzwi odblokowane';
	VIS.AStInformationDescription[0].wsDescription		:=	"";	 // Opis nie tłumaczony
	AudiInformationDescriptionIDTemp[0]					:=	1;
	
	AbInformationOnTemp[1]								:=	VIS.bConfectionEnding;
	VIS.AsInformationDescription[1]						:=	'Koniec konfekcji';
	VIS.AStInformationDescription[1].wsDescription		:=	"";	 // Opis nie tłumaczony
	AudiInformationDescriptionIDTemp[1]					:=	2;
	
	IF NOT VIS.bDispencersCatchEnableShow AND NOT VIS.bConfectionEnding THEN
		AbInformationOnTemp[2]							:=	NOT VIS.bDispencersCatchEnableShow;
		VIS.AsInformationDescription[2]					:=	'UWAGA! Włączony tryb słoików, chwytaki dozowanika wyłączone';
		VIS.AStInformationDescription[2].wsDescription	:=	"";	 // Opis nie tłumaczony
		AudiInformationDescriptionIDTemp[2]				:=	3;
	ELSE
		AbInformationOnTemp[2]	:=	FALSE;	
	END_IF
	
	AbInformationOnTemp[3]								:=	FALSE;//P00_PackML.fbPMLAuto.ePMLState = E_PMLState.ePMLState_IDLE AND bHomingCanceled;
	VIS.AsInformationDescription[3]						:=	'Anulowano bazowanie, naciśnij STOP i zbazuj stację';
	VIS.AStInformationDescription[3].wsDescription		:=	"";	 // Opis nie tłumaczony
	AudiInformationDescriptionIDTemp[3]					:=	4;
		
	AbInformationOnTemp[4]								:=	FALSE;//NOT P00_PackML.bFirstPositioningDone;
	VIS.AsInformationDescription[4]						:=	'Nie wykonano pierwszego bazowania po uruchomieniu';
	VIS.AStInformationDescription[4].wsDescription		:=	"";	 // Opis nie tłumaczony
	AudiInformationDescriptionIDTemp[4]					:=	5;
								
	AbInformationOnTemp[5]								:=	tonNoFormsBeforeDispencers.Q;
	VIS.AsInformationDescription[5]						:=	'Czekanie na formatki przed dozownikami';
	VIS.AStInformationDescription[5].wsDescription		:=	"";	 // Opis nie tłumaczony
	AudiInformationDescriptionIDTemp[5]					:=	6;            
	
	MAIN.tWeightTime;
	sWeightTime	:= 	Concat	(
					Concat	('/',
								INT_TO_STRING(LREAL_TO_INT(FLOOR(TIME_TO_LREAL(MAIN.tWeightTime)/1000.0)))),
							's'
							);		
					
	AbInformationOnTemp[6]								:=	VIS.bWeighingForm;
	VIS.AsInformationDescription[6]						:=	CONCAT('Trwa przeważanie formatek ',CONCAT(INT_TO_STRING(LREAL_TO_INT(FLOOR(TIME_TO_LREAL(MAIN.tonWeighingForm.ET)/1000.0))),sWeightTime));	
	VIS.AStInformationDescription[6].wsDescription		:=	WCONCAT("",WCONCAT(INT_TO_WSTRING(LREAL_TO_INT(FLOOR(TIME_TO_LREAL(MAIN.tonWeighingForm.ET)/1000.0))),STRING_TO_WSTRING(sWeightTime)));	
	AudiInformationDescriptionIDTemp[6]					:=	7;        
	
	AbInformationOnTemp[7]								:=	bHomingCanceled;
	VIS.AsInformationDescription[7]						:=	'Anulowano bazowanie - wybierz recepturę';
	VIS.AStInformationDescription[7].wsDescription		:=	"";	 // Opis nie tłumaczony
	AudiInformationDescriptionIDTemp[7]					:=	8;      
	
	AbInformationOnTemp[8]								:=	P02_Dispencers.tonTank1LevelWarning.Q;
	VIS.AsInformationDescription[8]						:=	'Niski poziom w zbiorniku 1';
	VIS.AStInformationDescription[8].wsDescription		:=	"";	 // Opis nie tłumaczony
	AudiInformationDescriptionIDTemp[8]					:=	9;    
	
	AbInformationOnTemp[9]								:=	P02_Dispencers.tonTank2LevelWarning.Q;
	VIS.AsInformationDescription[9]						:=	'Niski poziom w zbiorniku 2';
	VIS.AStInformationDescription[9].wsDescription		:=	"";	 // Opis nie tłumaczony
	AudiInformationDescriptionIDTemp[9]					:=	10;   
	
	AbInformationOnTemp[10]								:=	VIS.bCapSorterEmptyingMode;		
	VIS.AsInformationDescription[10]					:=	'Tryb opróżniania sortera nasadek';
	VIS.AStInformationDescription[10].wsDescription		:=	"";	 // Opis nie tłumaczony
	AudiInformationDescriptionIDTemp[10]				:=	11;   
	
	AbInformationOnTemp[11]								:=	VIS.bBottleSorterEmptyingMode;	
	VIS.AsInformationDescription[11]					:=	'Tryb opróżniania sortera butelek';
	VIS.AStInformationDescription[11].wsDescription		:=	"";	 // Opis nie tłumaczony
	AudiInformationDescriptionIDTemp[11]				:=	12;   
	
	AbInformationOnTemp[12]								:=	NOT P00_PackML.tonLongDelayAfterStart.Q AND P00_PackML.fbPMLAuto.ePMLState = E_PMLState.ePMLState_EXECUTE;	
	VIS.AsInformationDescription[12]					:=	CONCAT('',CONCAT(INT_TO_STRING(LREAL_TO_INT(FLOOR(TIME_TO_LREAL(P00_PackML.tonLongDelayAfterStart.ET)/1000.0))),'/40s'));	
	VIS.AStInformationDescription[12].wsDescription		:=	WCONCAT("",WCONCAT(INT_TO_WSTRING(LREAL_TO_INT(FLOOR(TIME_TO_LREAL(P00_PackML.tonLongDelayAfterStart.ET)/1000.0))),"/40s"));		
	AudiInformationDescriptionIDTemp[12]				:=	13;   
	
	AbInformationOnTemp[13]								:=	P00_PackML.tonCycleBadBottleConveyorFullSensor.Q;
	VIS.AsInformationDescription[13]					:=	'Odrzut - opróźnij';
	VIS.AStInformationDescription[13].wsDescription		:=	"";	 // Opis nie tłumaczony
	AudiInformationDescriptionIDTemp[13]				:=	14;   
	
	AbInformationOnTemp[14]								:=	NOT P00_PackML.tonbFirstCycle.Q;
	VIS.AsInformationDescription[14]					:=	'Trwa uruchamianie';
	VIS.AStInformationDescription[14].wsDescription		:=	"";	 // Opis nie tłumaczony
	AudiInformationDescriptionIDTemp[14]				:=	15;   
	
	AbInformationOnTemp[15]								:=	MAIN.bRFIDWeightShowAverageError;
	VIS.AsInformationDescription[15]					:=	'Zrób przeważanie (zbyt różna waga(<>40g) jednej z formatek od średniej)';
	VIS.AStInformationDescription[15].wsDescription		:=	"";	 // Opis nie tłumaczony	
	AudiInformationDescriptionIDTemp[15]				:=	16;   
	
	AbInformationOnTemp[16]								:=	VIS.bBottleTransferAllFormsToLabeler;
	VIS.AsInformationDescription[16]					:=	'Przenoszenie wszystkich opak. na etykieciarkę';
	VIS.AStInformationDescription[16].wsDescription		:=	"";	 // Opis nie tłumaczony
	AudiInformationDescriptionIDTemp[16]				:=	17;   
	
	AbInformationOnTemp[17]								:=	VIS.bBottleTransferAllFormsToExit;
	VIS.AsInformationDescription[17]					:=	'Przenoszenie wszystkich opak. na odrzut';
	VIS.AStInformationDescription[17].wsDescription		:=	"";	 // Opis nie tłumaczony	
	AudiInformationDescriptionIDTemp[17]				:=	18;   
	
	AbInformationOnTemp[18]								:=	IbEmergencyStop AND NOT IbBottleFeederSafety AND bBottleFeederEnable;
	VIS.AsInformationDescription[18]					:=	'Zamknij drzwi podajnika butelek';
	VIS.AStInformationDescription[18].wsDescription		:=	"RBI";	 // Opis nie tłumaczony	
	AudiInformationDescriptionIDTemp[18]				:=	19;   
	
	AbInformationOnTemp[19]								:=	bExEnable;
	VIS.AsInformationDescription[19]					:=	'Wlaczony tryb Ex';
	IF NOT P20_ExhaustFan.IbExhaustSystemReady THEN 
		VIS.AStInformationDescription[19].wsDescription		:=	"Nie gotowy-trwa rozruch";
		//VIS.AStInformationDescription[19].wsDescription		:=	"";//WConcat(UDINT_TO_WSTRING(VIS.udiExhaustFanVelocityCV),"rpm-EX");	 // Opis nie tłumaczony	
	ELSE
		VIS.AStInformationDescription[19].wsDescription		:=	"Gotowy";
	END_IF
	AudiInformationDescriptionIDTemp[19]				:=	20;   
	
	AbInformationOnTemp[20]								:=	VIS.bExEnableShow AND NOT bExEnable;
	VIS.AsInformationDescription[20]					:=	'Receptura ma włączony tryb EX-przekręć (koło panelu i na scianie), sprawdź czujnik poziomu';
	VIS.AStInformationDescription[20].wsDescription		:=	"?EX?";	 // Opis nie tłumaczony	
	AudiInformationDescriptionIDTemp[20]				:=	21;   

	AbInformationOnTemp[21]								:=	NOT bTank1SupplyPumpEnable;
	VIS.AsInformationDescription[21]					:=	'Pompa wyłączona';
	VIS.AStInformationDescription[21].wsDescription		:=	"";	 // Opis nie tłumaczony	
	AudiInformationDescriptionIDTemp[21]				:=	22;   

	AbInformationOnTemp[22]								:=	P16_LabelMachine.tonLabelMachineFullSensorInfo.Q;
	VIS.AsInformationDescription[22]					:=	'Kolejka - etykieciarka';
	VIS.AStInformationDescription[22].wsDescription		:=	"ETK";	 // Opis nie tłumaczony	
	AudiInformationDescriptionIDTemp[22]				:=	23;   
	
	AbInformationOnTemp[23]								:=	P10_GripperScrewer.bGripperScrewer1ChangeRubbers;
	VIS.AsInformationDescription[23]					:=	'Zakręcarka 1 - zmień gumy';
	VIS.AStInformationDescription[23].wsDescription		:=	"Z1";	 // Opis nie tłumaczony	
	AudiInformationDescriptionIDTemp[23]				:=	24;   
		
	AbInformationOnTemp[24]								:=	P10_GripperScrewer.bGripperScrewer2ChangeRubbers;
	VIS.AsInformationDescription[24]					:=	'Zakręcarka 2 - zmień gumy';
	VIS.AStInformationDescription[24].wsDescription		:=	"Z2";	 // Opis nie tłumaczony	
	AudiInformationDescriptionIDTemp[24]				:=	25;   


	(**KROK 3**)
	(**Dodawanie komunikatów**)
	VIS.iActiveInformation := 0;
	FOR i := 0 TO 63-1 DO
		IF AbInformationOnTemp[i] THEN
			VIS.AsInformationDescription[i]			:=	VIS.AsInformationDescription[i];
			VIS.AStInformationDescription[i].udiID  :=	AudiInformationDescriptionIDTemp[i];
			VIS.iActiveInformation					:=	VIS.iActiveInformation	+ 1;
		ELSE
			VIS.AsInformationDescription[i]			:= '';
			VIS.AStInformationDescription[i].udiID 	:= 0;
		END_IF
	END_FOR
	
	(**KROK 4**)
	(**Sortowanie tablicy**)
	n := 63;
	WHILE n>1 DO
		FOR i := 0 TO 63-1 DO
			IF VIS.AsInformationDescription[i] = '' THEN //Jeżeli pusty
				VIS.AsInformationDescription[i]		:=	VIS.AsInformationDescription[i+1];
				VIS.AsInformationDescription[i+1]	:=	'';
			END_IF
			IF VIS.AStInformationDescription[i].udiID = 0 THEN //Jeżeli pusty
				VIS.AStInformationDescription[i].udiID				:=	VIS.AStInformationDescription[i+1].udiID;
				VIS.AStInformationDescription[i].wsDescription		:=	VIS.AStInformationDescription[i+1].wsDescription;			
				VIS.AStInformationDescription[i+1].udiID			:=	0;
				VIS.AStInformationDescription[i+1].wsDescription	:=	"";			
			END_IF		
		END_FOR
		n := n - 1;
	END_WHILE
	
	
	(*Wykrywanie nowego ostrzezenia do wizualizacji*)
	
	
	
	rtInformationNew ( CLK:= iAbInformationOnTempCounterTemp	<> VIS.iActiveInformation AND VIS.iActiveInformation > 0);
	iAbInformationOnTempCounterTemp	:=	VIS.iActiveInformation;
	IF rtInformationNew.Q THEN
		VIS.bInformationNew	:=	TRUE;
	END_IF
	tonInformationNew (IN:= VIS.bInformationNew ,PT:=T#1S);
	IF tonInformationNew.Q THEN
		VIS.bInformationNew	:=	FALSE;
	END_IF
	(*Koniec Wykrywanie nowego ostrzezenia do wizualizacji*)
	
	VIS.AStInformationDescription[0].udiID;VIS.AStInformationDescription[0].wsDescription;
	VIS.AStInformationDescription[1].udiID;VIS.AStInformationDescription[1].wsDescription;
	VIS.AStInformationDescription[2].udiID;VIS.AStInformationDescription[2].wsDescription;
	VIS.AStInformationDescription[3].udiID;VIS.AStInformationDescription[3].wsDescription;
//END_IF
END_ACTION

END_PROGRAM

// ---- POUs/P07_ROPP.TcPOU
(*
Nazwa:			P07_ROPP
Opis:			ROPP
Wersja:			v0.1
Data:			2025-02-07
Autor:			DP
Urzadzenia:		
Konfiguracja:	
Info:
- 
*)
PROGRAM P07_ROPP
VAR_INPUT
	//Spowalniacz	
	//...
	
	//Podajnik
	//...
	
	//Sprawdzanie nasadek
	
	//Stoper
	
	//Przeciaganie

	//Zakrecanie
	//..

	//Sprawdzanie zakrecenia
END_VAR
VAR
	(*****************SPOWALNIACZ*******************)
	fbROPPSlower										: FB_MitsubishiInverter;
	eROPPSlowerState									: E_Station;			
	eROPPSlowerRunningState								: E_ConveyorState;	
	fbROPPSlowerState									: FB_State;		
	QnROPPSlowerVelocitySV 								AT %Q*: UDINT; 			// Nastawa prędkości transportera
	InROPPSlowerVelocityCV 								AT %I*: UDINT;
	InROPPSlowerSTW 									AT %I*: UINT; 			// Statusword transportera wyjściowego
	QnROPPSlowerCTW 									AT %Q*: UINT;  			// Controlword transportera wyjsciowego
	InROPPSlowerErrorCode 								AT %I*:UINT;
	IbROPPSevenFormSensor 								: BOOL;		
	IbROPPBeforeSevenFormSensor 						: BOOL;		



	(*******************PODAJNIK*********************)
	fbROPPFeeder										: FB_ROPPFeeder;
	fbROPPFeederState									: FB_State;	
	eROPPFeederState									: E_Station;
	eROPPFeederRunningState								: E_CapFeederState; 	// Stan pracy 
	QbROPPFeederHeightUpCmd 							AT %Q*: BOOL; 			// Wyjście sterujące podnośnikiem podajnika nakrętek, Silnik w górę
	QbROPPFeederHeightDownCmd 							AT %Q*: BOOL; 			// Wyjście sterujące podnośnikiem podajnika nakrętek, Silnik w dół
	QudiROPPFeederHeightEncoderSetCV					AT %Q*: UDINT;			// Enkoder - Set Counter value
	QbROPPFeederHeightEncoderSetC						AT %Q*: BOOL; 			// Enkoder - Set Counter 
	IudiROPPFeederHeightEncoderCV 						AT %I*: UDINT;	 		// Enkoder - Counter value
	IbROPPFeederHeightEncoderSetCDone					AT %I*: BOOL; 			// Enkoder - Set Counter done
	QbROPPFeederSorterVibrator 							AT %Q*: BOOL; 			// Wyjście sterujące 
	QbROPPFeederSorterAir 								AT %Q*: BOOL; 			// Wyjście sterujące 
	QbROPPFeederConveyorStart 							AT %Q*: BOOL; 			// Wyjście sterujące 
	QbROPPFeederConveyorStop							AT %Q*: BOOL; 			// Wyjście sterujące 
	IbROPPFeederAirOK									: BOOL; 			
	IbROPPFeederCapsWheelLevel							: BOOL; 			
	IbROPPFeederCapsLevel								: BOOL; 			
	IbROPPFeederCapsSleeveUp							: BOOL; 
	QnROPPFeederSorterVelocitySV 						AT %Q*: UDINT; 			// Nastawa prędkości
	InROPPFeederSorterVelocityCV 						AT %I*: UDINT;		
	InROPPFeederSorterSTW 								AT %I*: UINT; 			// Statusword transportera wejściowo wyjściowego
	QnROPPFeederSorterCTW 								AT %Q*: UINT;  			// Controlword transportera we/wy
	IbROPPFeederSorterWcState							AT %I*: BOOL; 			// Statusword transportera wejściowo wyjściowego
	TimerROPPFeederEnable: TOF;
	rtROPPFeederEnable: R_TRIG;
	tonROPPFeederEnable: TON;

	(*******Sprawdzanie nasadek**********)
	fbIbROPPPuttedCheckSensor							: FB_InputFilter_v2;
	IbROPPPuttedCheckSensor 							: BOOL;			
	
	(*******STOPER**********)
	QbROPPStoperBeforeActuator							: BOOL;
	QbROPPStoperAfterActuator							: BOOL;
	bROPPStoperBeforeActuatorLastState					: BOOL;
	bROPPStoperAfterActuatorLastState					: BOOL;	
	fbROPPStoperSensorDelay								: FB_InputFilter;
	lrROPPStoperPosition								: LREAL;
	tofQbROPPStoperActuator								: TOF;
	
	(*******PRZECIAGANIE**********)
	fbROPPDrag											: FB_FormsDragStepper;
	eROPPDragState										: E_Station;					// Stan zakręcarki
	eROPPDragRunningState								: E_DragStationState;			// Stan zakręcarki
	fbROPPDragState										: FB_State;
	//WEJSCIA I WYJSCIA SPRZETOW
	QbROPPDragLeadBefore1Actuator        				: BOOL;				
	QbROPPDragActuator                	  				: BOOL;				
	IbROPPDragHomingSensor 								: BOOL;			// Czujnik bazowania	
	IbROPPDragLeadBefore1UpSensor 		 				: BOOL;			// Czujnik
	IbROPPDragLeadBefore2UpSensor 		 				: BOOL;			// Czujnik
	IbROPPDragUpSensor 			 						: BOOL;			// Czujnik
	IbROPPDragDownSensor 			 					: BOOL;			// Czujnik
	
	(*******ZAKRECANIE**********)
	fbROPPCapping										: FB_ROPPCapping;
	fbROPPCappingState									: FB_State;	
	eROPPCappingState									: E_Station;
	eROPPCappingRunningState							: E_GripperScrewer; 	// Stan pracy 
	QbROPPCappingHeightUpCmd 							AT %Q*: BOOL; 		
	QbROPPCappingHeightDownCmd 							AT %Q*: BOOL; 		
	QudiROPPCappingHeightEncoderSetCV					AT %Q*: UDINT;			// Enkoder - Set Counter value
	QbROPPCappingHeightEncoderSetC						AT %Q*: BOOL; 			// Enkoder - Set Counter 
	IudiROPPCappingHeightEncoderCV 						AT %I*: UDINT;	 		// Enkoder - Counter value
	IbROPPCappingHeightEncoderSetCDone					AT %I*: BOOL; 			// Enkoder - Set Counter done

	QbROPPCapping1Tool1Actuator							AT %Q*: BOOL; 	
	QbROPPCapping2Tool1Actuator 						AT %Q*: BOOL; 
	IbROPPCapping1Tool1ActuatorUpSensor					: BOOL; 
	IbROPPCapping1Tool1ActuatorDownSensor				: BOOL; 
	IbROPPCapping2Tool1ActuatorUpSensor					: BOOL; 
	IbROPPCapping2Tool1ActuatorDownSensor				: BOOL; 

	IbROPPCapping1Tool2ActuatorUpSensor					: BOOL; 
	IbROPPCapping1Tool2ActuatorCappingDoneSensor		: BOOL; 
	IbROPPCapping2Tool2ActuatorUpSensor					: BOOL; 
	IbROPPCapping2Tool2ActuatorCappingDoneSensor		: BOOL; 


	QbROPPCapping12Tool1BlockActuator 					AT %Q*: BOOL; 
	QbROPPCappingBlockActuator 							AT %Q*: BOOL; 
	
	QbROPPCapping1Tool2Down								: BOOL; 	
	QbROPPCapping1Tool2Tight							: BOOL; 	
	QbROPPCapping1Tool2Realese							: BOOL; 
	QbROPPCapping2Tool2Down								: BOOL; 	
	QbROPPCapping2Tool2Tight							: BOOL; 
	QbROPPCapping2Tool2Realese							: BOOL; 

	QbROPPCappingFormPositioning						AT %Q*: BOOL; 	
	IbROPPCappingFormPositioningOnSensor 			 	: BOOL;			// Czujnik
	IbROPPCappingFormPositioningOffSensor 			 	: BOOL;			// Czujnik
	
	QnROPPCapping1VelocitySV 							AT %Q*: UDINT; 		
	InROPPCapping1VelocityCV 							AT %I*: UDINT;		
	InROPPCapping1STW 									AT %I*: UINT; 			// Statusword transportera wejściowo wyjściowego
	QnROPPCapping1CTW 									AT %Q*: UINT;  			// Controlword transportera we/wy
	IbROPPCapping1WcState								AT %I*: BOOL; 			// Statusword transportera wejściowo wyjściowego
	QnROPPCapping2VelocitySV 							AT %Q*: UDINT; 		
	InROPPCapping2VelocityCV 							AT %I*: UDINT;		
	InROPPCapping2STW 									AT %I*: UINT; 			// Statusword transportera wejściowo wyjściowego
	QnROPPCapping2CTW 									AT %Q*: UINT;  			// Controlword transportera we/wy
	IbROPPCapping2WcState								AT %I*: BOOL; 			// Statusword transportera wejściowo wyjściowego

	TimerROPPCappingEnable: TOF;
	rtROPPCappingEnable: R_TRIG;
	tonROPPCappingEnable: TON;

	(*******Sprawdzanie zakręcenia**********)
	fbIbROPPCappingCheckSensor							: FB_InputFilter_v2;
	IbROPPCappingCheckSensor 							: BOOL;			// Czujnik 
	//IbROPPCappingCheckFormSensor						: BOOL;			// Czujnik 
	
	(*RFID*)
	//Przed
	bReadedCardBeforeROPP 								: BOOL;				
	nReadedCardBeforeROPP 								: ULINT;	
	fbBeforeROPPReader   								: FB_IfmIoLinkRfid;
	AusiBeforeROPPReaderInputData  						AT %I* : ARRAY[0..27] OF USINT;
	IbBeforeROPPReaderTagPresent						AT %I* : BOOL;
	IBBeforeROPPReaderErrorValue						AT %I* : BYTE;
	IbBeforeROPPReaderCmdEnd							AT %I* : BOOL;
	IBBeforeROPPReaderDataCounterIn						AT %I* : BYTE;
	IbBeforeROPPReaderCmdStartAck						AT %I* : BOOL;
	IbBeforeROPPReaderCmdStart							AT %Q* : BOOL;
	IBBeforeROPPReaderCmmandValue						AT %Q* : BYTE;
	IBBeforeROPPReaderDataCounterOut					AT %Q* : BYTE;
	AusiBeforeROPPReaderOutputData  					AT %Q* : ARRAY[0..27] OF USINT;	
	//Za
	bReadedCardAfterROPP 								: BOOL;				
	nReadedCardAfterROPP 								: ULINT;	
	fbAfterROPPReader   								: FB_IfmIoLinkRfid;
	AusiAfterROPPReaderInputData  						AT %I* : ARRAY[0..27] OF USINT;
	IbAfterROPPReaderTagPresent							AT %I* : BOOL;
	IBAfterROPPReaderErrorValue							AT %I* : BYTE;
	IbAfterROPPReaderCmdEnd								AT %I* : BOOL;
	IBAfterROPPReaderDataCounterIn						AT %I* : BYTE;
	IbAfterROPPReaderCmdStartAck						AT %I* : BOOL;
	IbAfterROPPReaderCmdStart							AT %Q* : BOOL;
	IBAfterROPPReaderCmmandValue						AT %Q* : BYTE;
	IBAfterROPPReaderDataCounterOut						AT %Q* : BYTE;
	AusiAfterROPPReaderOutputData  						AT %Q* : ARRAY[0..27] OF USINT;	

	(*Lampy*)
	QiROPPRedSignalizationLamp 							AT %Q* : INT;				
	QiROPPGreenSignalizationLamp 						AT %Q* : INT;					
	QiROPPBlueSignalizationLamp 						AT %Q* : INT;				
	QiROPPWhiteSignalizationLamp 						AT %Q* : INT;				
	QbROPPStartLamp			 							AT %Q* : BOOL;				// Sygnalizacja startu cyklu poprzez lampkę na przyciskac
	QbROPPResetLamp 									AT %Q* : BOOL; 				// Sygnalizacja Resetu bezpieczeństwa poprzez lampkę naprzycisku reset

	(*Przyciski*)
	IbROPPCycleStartButton								AT %I* :BOOL;		//Przycisk Startu cyklu
	//IbSafetyResetIn									AT %I* :BOOL;		//Reset
	IbROPPCycleStopButton								AT %I* :BOOL;		//Przycisk Stopu cyklu

	(*Safety*)
	IbROPPEmergencyStopButton0Pressed					AT %I* :BOOL;		
	IbROPPEmergencyStopButton1Pressed					AT %I* :BOOL;		
	IbROPP0DoorsOpen 									AT %I* :BOOL;		
	IbROPP1DoorsOpen									AT %I* :BOOL;		

	QbROPPDoors0Close									AT %Q* :BOOL;		// Rozkaz zamkniecia 
	QbROPPDoors1Close									AT %Q* :BOOL;		// Rozkaz zamkniecia 
	
	(*Zawór główny*)
	QbROPPCompressedAir								AT %Q*		:BOOL;		
	IbROPPCompressedAirOK 							AT %I*		:BOOL;		//Zasilanie powietrzem sprężonym OK	
	
	(*Zasilanie*)
	IbROPPFuseFB1OK										AT %I* :BOOL;		//		
	IbROPPFuseFB2OK										AT %I* :BOOL;		//	
	IbROPPFuseFB3OK										AT %I* :BOOL;		//	
	IbROPPFuseFB4OK										AT %I* :BOOL;		//	
	IbROPPFuseFB5OK										AT %I* :BOOL;		//	
	IbROPPFuseFB6OK										AT %I* :BOOL;		//	
	IbROPPFuseFB7OK										AT %I* :BOOL;		//	
	IbROPPFuseFB8OK										AT %I* :BOOL;		//		
	IbROPPFuseFB9OK										AT %I* :BOOL;		//		
	
	(*DI wyspy pneumatycznej*)
	QABPneumaticROPPEB1ValveCoils 						AT %Q* 	: ARRAY[1..5] OF BYTE;	
	IABPneumaticROPPEB1DigitalInput 					AT %I* 	: ARRAY[1..4] OF BYTE;
	IuiPneumaticROPPEB1State							AT %I* 	: UINT;	

	(*Czujniki formatek*)
	IbROPPThirdFormSensor	 							: BOOL; 		// Czujnik dojazdu 3 formatki
	IbROPPAfterFormSensor								: BOOL;			// Czujnik za stacją			
	IbROPPAfter2FormSensor								: BOOL;			// Czujnik 2 formatek za stacją
	IbROPPAfter3FormSensor								: BOOL;			// Czujnik 2 formatek za stacją
	
	(*Manual*)
	rtManualMode										: R_TRIG;
	ftManualMode										: F_TRIG;
	
	(****Inne***)
	bTemp												: BOOL;
	bConveyorTest1										: BOOL;
	bROPPFeederRunTest									: BOOL;
	rtQbROPPStoperBeforeActuator						: R_TRIG;
	tonQbROPPStoperBeforeActuator						: TON;	
	rtQbROPPStoperAfterActuator							: R_TRIG;
	tonQbROPPStoperAfterActuator						: TON;
	tonQbROPPStoperBeforeActuatorOn						: TON;
	
END_VAR

aPowerSupply();
aButtons();
aPneumatics();
aRFID();
aRFID_FB();
aSafety();
aSignalization();
aLimits();
a1_Slower();
a2_Feeder();
a3_PuttedCheck();
a4_Stoper();
a5_Draging();
//a6_Capping();
a7_CappingCheck();

(*BAZOWANIE - ZMIAN*)
//Spowalniacz
//...
//Podajnik
tonROPPFeederEnable (IN:=bROPPFeederEnable,PT:=T#5S); 
rtROPPFeederEnable(CLK:=tonROPPFeederEnable.Q,Q=>);
IF rtROPPFeederEnable.Q AND (P00_PackML.fbPMLAuto.ePMLState = E_PMLState.ePMLState_IDLE OR P00_PackML.fbPMLAuto.ePMLState = E_PMLState.ePMLState_EXECUTE)   THEN
	VIS_ROPP.bROPPFeederHeightSet:=TRUE;
ELSIF fbROPPFeeder.eState=E_Station.eHomingDone	OR	VIS.bErrorOccure THEN
 	VIS_ROPP.bROPPFeederHeightSet:=FALSE;
END_IF
//Sprawdzanie nasadek
//..
//Przeciaganie
//...
//Zakrecanie
tonROPPCappingEnable (IN:=bROPPCappingEnable,PT:=T#5S); 
rtROPPCappingEnable(CLK:=tonROPPCappingEnable.Q,Q=>);
IF rtROPPCappingEnable.Q AND (P00_PackML.fbPMLAuto.ePMLState = E_PMLState.ePMLState_IDLE OR P00_PackML.fbPMLAuto.ePMLState = E_PMLState.ePMLState_EXECUTE)   THEN
	VIS_ROPP.bROPPCappingHeightSet:=TRUE;
ELSIF fbROPPCapping.eState=E_Station.eHomingDone	OR	VIS.bErrorOccure THEN
 	VIS_ROPP.bROPPCappingHeightSet:=FALSE;
END_IF
//Sprawdzanie zakręcenia
//..
(*KONIEC BAZOWANIE - ZMIANA*)

(*Opoznienie wyłączanie enabla*)
//Spowalniacz
//..
//Podajnik
TimerROPPFeederEnable	(IN:=bROPPFeederEnable,	PT:=T#2S);
//Sprawdzanie nasadek
//..
//Przeciaganie
//...
//Zakrecanie
TimerROPPCappingEnable	(IN:=bROPPCappingEnable, PT:=T#2S);
//Sprawdzanie zakręcenia
//..

(*Staty*)
//Spowalniacz
//...
//Podajnik
fbROPPFeederState(
	eState							:=	eROPPFeederState , 
	bRun							:=	VIS_ROPP.bROPPFeederRun,	
	eCapFeederRunningState			:=	eROPPFeederRunningState , 
	sStateDesc						=>	VIS_ROPP.sROPPFeederState,
	iState							=>	VIS_ROPP.iROPPFeederState);	
//Sprawdzanie nasadek
//..
//Przeciaganie
fbROPPDragState(
	eState							:= eROPPDragState , 
	bRun							:= VIS_ROPP.bROPPDragRun,	
	eFormsDragingRunningState		:= eROPPDragRunningState , 
	sStateDesc						=> VIS_ROPP.sROPPDragState,
	iState							=> VIS_ROPP.iROPPDragState);	
//Zakrecanie
fbROPPCappingState(
	eState							:=	eROPPCappingState , 
	bRun							:=	VIS_ROPP.bROPPCappingRun1 OR VIS_ROPP.bROPPCappingRun2,	
	eGripperScrewerRunningState		:=	eROPPCappingRunningState , 
	sStateDesc						=>	VIS_ROPP.sROPPCappingState,
	iState							=>	VIS_ROPP.iROPPCappingState);	
//Sprawdzanie zakręcenia
//..

(********KASOWANIE ROZKAZÓW CYKLI*********)
//Spowalniacz
//...
//Podajnik
//...
//Sprawdzanie nasadek
//..
//Przeciaganie
IF fbROPPDrag.bCycleDone AND bManualMode THEN
	VIS_ROPP.bROPPDragRun 				:= FALSE;
	GVL_ROPP.bROPPDragPrepareRun		:= FALSE;
END_IF
//Zakrecanie
IF fbROPPCapping.bCycleDone1 AND bManualMode THEN
	VIS_ROPP.bROPPCappingRun1 				:= FALSE;
END_IF
IF fbROPPCapping.bCycleDone2 AND bManualMode THEN
	VIS_ROPP.bROPPCappingRun2 				:= FALSE;
END_IF
//Sprawdzanie zakręcenia
//..

ACTION a1_Slower:
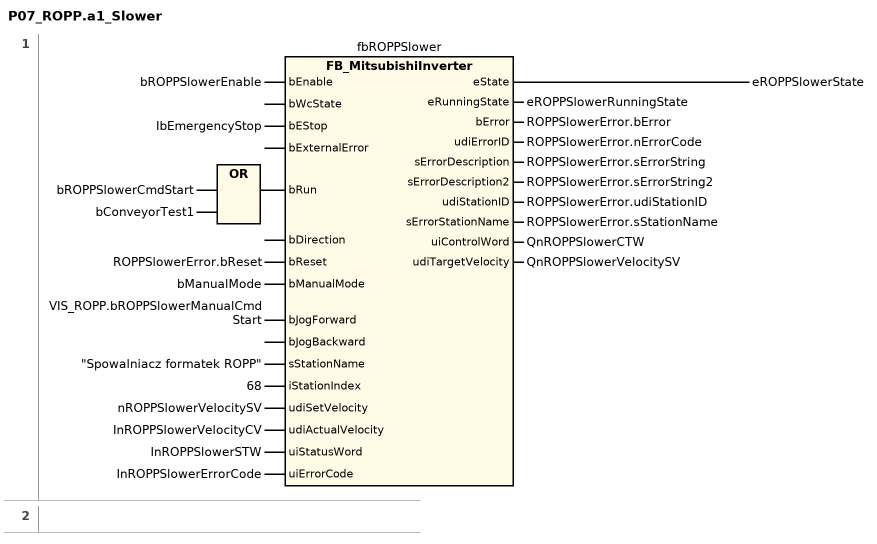
// NETWORK 1
fbROPPSlower(
    bEnable := bROPPSlowerEnable,
    bEStop := IbEmergencyStop,
    bRun := bROPPSlowerCmdStart OR bConveyorTest1,
    bReset := ROPPSlowerError.bReset,
    bManualMode := bManualMode,
    bJogForward := VIS_ROPP.bROPPSlowerManualCmdStart,
    sStationName := "Spowalniacz formatek ROPP",
    iStationIndex := 68,
    udiSetVelocity := nROPPSlowerVelocitySV,
    udiActualVelocity := InROPPSlowerVelocityCV,
    uiStatusWord := InROPPSlowerSTW,
    uiErrorCode := InROPPSlowerErrorCode,
    eRunningState => eROPPSlowerRunningState,
    bError => ROPPSlowerError.bError,
    udiErrorID => ROPPSlowerError.nErrorCode,
    sErrorDescription => ROPPSlowerError.sErrorString,
    sErrorDescription2 => ROPPSlowerError.sErrorString2,
    udiStationID => ROPPSlowerError.udiStationID,
    sErrorStationName => ROPPSlowerError.sStationName,
    uiControlWord => QnROPPSlowerCTW,
    udiTargetVelocity => QnROPPSlowerVelocitySV); // FB_MitsubishiInverter
eROPPSlowerState := fbROPPSlower.eState;

// NETWORK 2
END_ACTION

ACTION a2_Feeder:
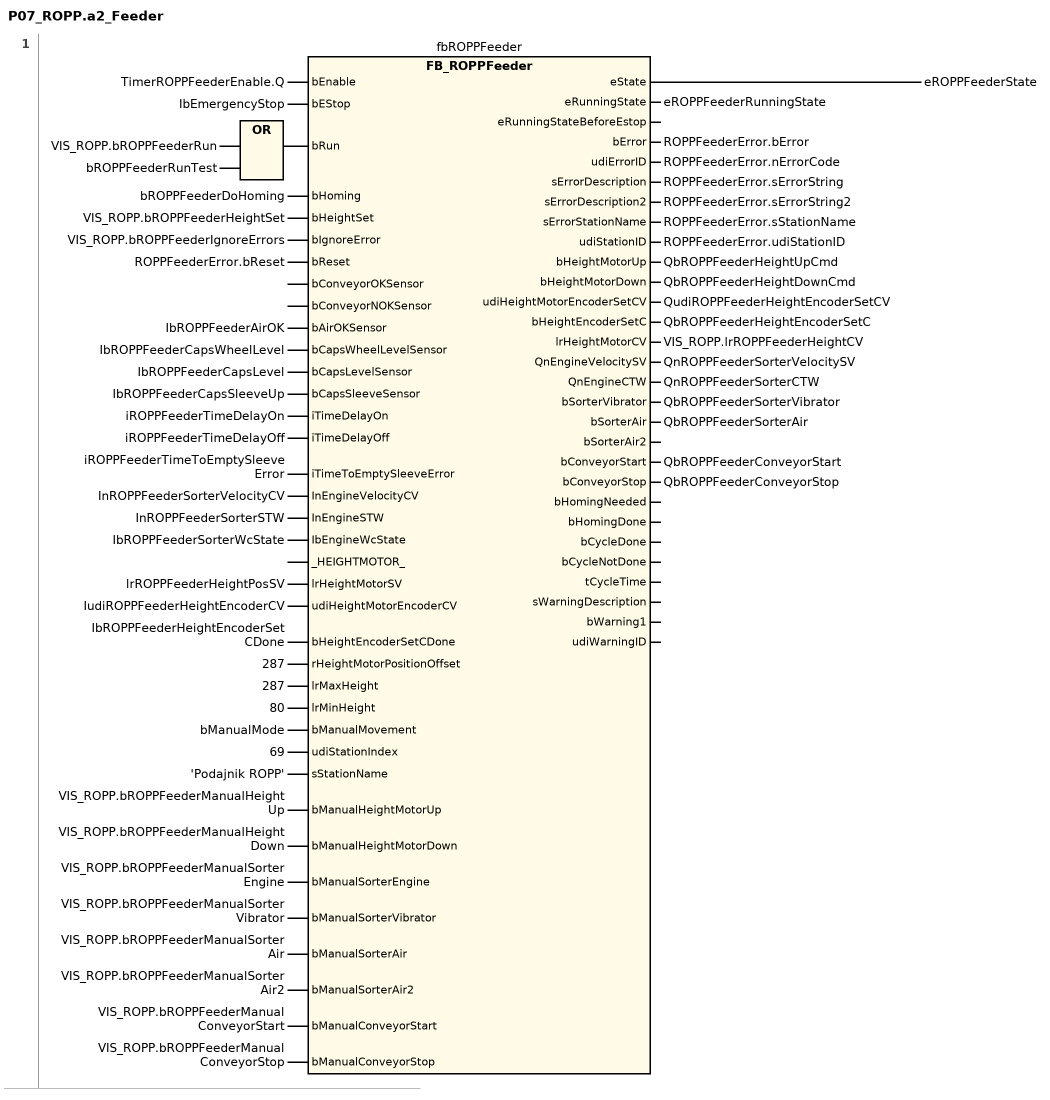
// NETWORK 1
fbROPPFeeder(
    bEnable := TimerROPPFeederEnable.Q,
    bEStop := IbEmergencyStop,
    bRun := VIS_ROPP.bROPPFeederRun OR bROPPFeederRunTest,
    bHoming := bROPPFeederDoHoming,
    bHeightSet := VIS_ROPP.bROPPFeederHeightSet,
    bIgnoreError := VIS_ROPP.bROPPFeederIgnoreErrors,
    bReset := ROPPFeederError.bReset,
    bAirOKSensor := IbROPPFeederAirOK,
    bCapsWheelLevelSensor := IbROPPFeederCapsWheelLevel,
    bCapsLevelSensor := IbROPPFeederCapsLevel,
    bCapsSleeveSensor := IbROPPFeederCapsSleeveUp,
    iTimeDelayOn := iROPPFeederTimeDelayOn,
    iTimeDelayOff := iROPPFeederTimeDelayOff,
    iTimeToEmptySleeveError := iROPPFeederTimeToEmptySleeveError,
    InEngineVelocityCV := InROPPFeederSorterVelocityCV,
    InEngineSTW := InROPPFeederSorterSTW,
    IbEngineWcState := IbROPPFeederSorterWcState,
    lrHeightMotorSV := lrROPPFeederHeightPosSV,
    udiHeightMotorEncoderCV := IudiROPPFeederHeightEncoderCV,
    bHeightEncoderSetCDone := IbROPPFeederHeightEncoderSetCDone,
    rHeightMotorPositionOffset := 287,
    lrMaxHeight := 287,
    lrMinHeight := 80,
    bManualMovement := bManualMode,
    udiStationIndex := 69,
    sStationName := 'Podajnik ROPP',
    bManualHeightMotorUp := VIS_ROPP.bROPPFeederManualHeightUp,
    bManualHeightMotorDown := VIS_ROPP.bROPPFeederManualHeightDown,
    bManualSorterEngine := VIS_ROPP.bROPPFeederManualSorterEngine,
    bManualSorterVibrator := VIS_ROPP.bROPPFeederManualSorterVibrator,
    bManualSorterAir := VIS_ROPP.bROPPFeederManualSorterAir,
    bManualSorterAir2 := VIS_ROPP.bROPPFeederManualSorterAir2,
    bManualConveyorStart := VIS_ROPP.bROPPFeederManualConveyorStart,
    bManualConveyorStop := VIS_ROPP.bROPPFeederManualConveyorStop,
    eRunningState => eROPPFeederRunningState,
    bError => ROPPFeederError.bError,
    udiErrorID => ROPPFeederError.nErrorCode,
    sErrorDescription => ROPPFeederError.sErrorString,
    sErrorDescription2 => ROPPFeederError.sErrorString2,
    sErrorStationName => ROPPFeederError.sStationName,
    udiStationID => ROPPFeederError.udiStationID,
    bHeightMotorUp => QbROPPFeederHeightUpCmd,
    bHeightMotorDown => QbROPPFeederHeightDownCmd,
    udiHeightMotorEncoderSetCV => QudiROPPFeederHeightEncoderSetCV,
    bHeightEncoderSetC => QbROPPFeederHeightEncoderSetC,
    lrHeightMotorCV => VIS_ROPP.lrROPPFeederHeightCV,
    QnEngineVelocitySV => QnROPPFeederSorterVelocitySV,
    QnEngineCTW => QnROPPFeederSorterCTW,
    bSorterVibrator => QbROPPFeederSorterVibrator,
    bSorterAir => QbROPPFeederSorterAir,
    bConveyorStart => QbROPPFeederConveyorStart,
    bConveyorStop => QbROPPFeederConveyorStop); // FB_ROPPFeeder
eROPPFeederState := fbROPPFeeder.eState;
END_ACTION

ACTION a3_PuttedCheck:

fbIbROPPPuttedCheckSensor(bIN:= IbROPPPuttedCheckSensor, tFilterTimeOn:=T#0MS , tFilterTimeOff:= T#0MS, bOUT=> );
fbIbROPPPuttedCheckSensor.bOUT;


IbROPPSevenFormSensor;

//Wizka
VIS_ROPP.bROPPPuttedCheckOK	:=	fbIbROPPPuttedCheckSensor.bOUT;
END_ACTION

ACTION a4_Stoper:
(*****STOPER PRZED STACJĄ***********)
QbROPPStoperBeforeActuator;									   					  					   
lrROPPStoperPosition	:=	(188.25 * EXPT(lrROPPDragVelocity,-0.404));
rtQbROPPStoperBeforeActuator	(CLK:= 	fbROPPDrag.lrActualDragPosition > (lrROPPStoperPosition) AND 
								fbROPPDrag.lrActualDragPosition < 100 AND VIS_ROPP.bROPPDragRun AND
								fbROPPDrag.eRunningState = E_DragStationState.eDraging AND
						   ((P00_PackML.fbPMLAuto.ePMLState = E_PMLState.ePMLState_STOPPING) OR  (P00_PackML.fbPMLAuto.ePMLState = E_PMLState.ePMLState_EXECUTE))
						,Q=>);	
//tonQbROPPStoperBeforeActuator	(IN:=QbROPPStoperBeforeActuator, PT:=T#80MS);		//bylo 120	
tonQbROPPStoperBeforeActuatorOn	(IN:=QbROPPStoperBeforeActuator AND bFormTransportersBeforeROPPCmdStart , PT:=T#150MS);	
tonQbROPPStoperBeforeActuator	(IN:=tonQbROPPStoperBeforeActuatorOn.Q (*AND P07_ROPP.IbROPPThirdFormSensor*), PT:=T#0MS);			
IF rtQbROPPStoperBeforeActuator.Q THEN
	QbROPPStoperBeforeActuator	:=	TRUE;
END_IF
IF tonQbROPPStoperBeforeActuator.Q THEN
	QbROPPStoperBeforeActuator	:=	FALSE;
END_IF
(*****KONIEC STOPER PRZED STACJĄ***********)

(*****STOPER ZA STACJĄ***********)
QbROPPStoperAfterActuator;									   					  					   
lrROPPStoperPosition	:=	(188.25 * EXPT(lrROPPDragVelocity,-0.404));
rtQbROPPStoperAfterActuator	(CLK:= 	fbROPPDrag.lrActualDragPosition > 100 AND 
								fbROPPDrag.lrActualDragPosition < 120 AND VIS_ROPP.bROPPDragRun AND
								fbROPPDrag.eRunningState = E_DragStationState.eDraging AND
								P15_FormTransporters.eFormTransporterScrewerRunningState = E_ConveyorState.eWorking AND
						   ((P00_PackML.fbPMLAuto.ePMLState = E_PMLState.ePMLState_STOPPING) OR  (P00_PackML.fbPMLAuto.ePMLState = E_PMLState.ePMLState_EXECUTE))
						,Q=>);	
tonQbROPPStoperAfterActuator	(IN:=QbROPPStoperAfterActuator, PT:=T#260MS);					
IF rtQbROPPStoperAfterActuator.Q THEN
	QbROPPStoperAfterActuator	:=	TRUE;
END_IF
IF tonQbROPPStoperAfterActuator.Q THEN
	QbROPPStoperAfterActuator	:=	FALSE;
END_IF
(*****KONIEC STOPER ZA STACJĄ***********)


//Manual
rtManualMode	(CLK:=bManualMode,	Q=>);
ftManualMode	(CLK:=bManualMode,	Q=>);
IF rtManualMode.Q THEN
	bROPPStoperBeforeActuatorLastState	:=	QbROPPStoperBeforeActuator;
	bROPPStoperBeforeManualActuator		:=	QbROPPStoperBeforeActuator;
	bROPPStoperAfterActuatorLastState	:=	QbROPPStoperAfterActuator;
	bROPPStoperAfterManualActuator		:=	QbROPPStoperAfterActuator;
END_IF
IF bManualMode THEN
	QbROPPStoperBeforeActuator			:=	bROPPStoperBeforeManualActuator;
	QbROPPStoperAfterActuator			:=	bROPPStoperAfterManualActuator;
END_IF
IF ftManualMode.Q THEN
	QbROPPStoperBeforeActuator			:= bROPPStoperBeforeActuatorLastState;
	QbROPPStoperAfterActuator			:= bROPPStoperAfterActuatorLastState;
END_IF
// Koniec Manual
END_ACTION

ACTION a5_Draging:
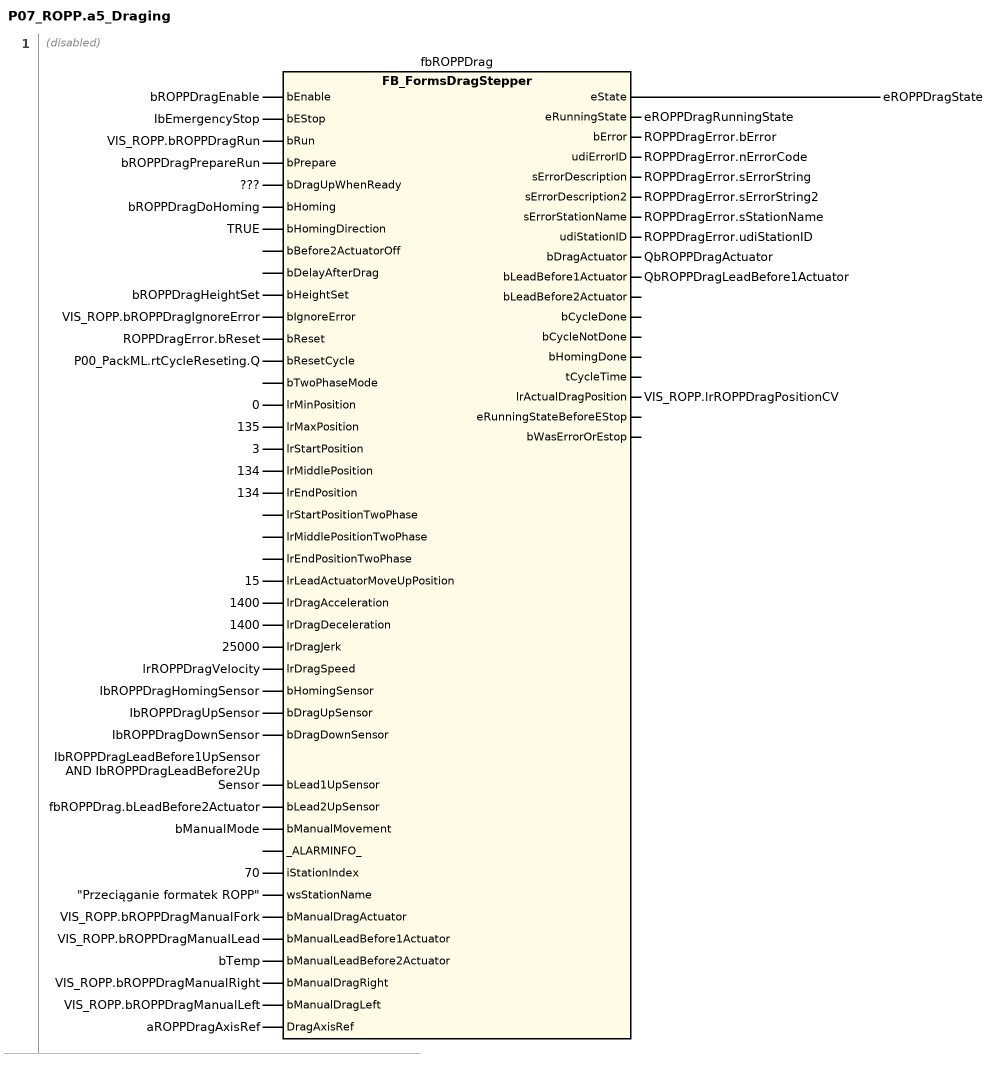
// NETWORK 1 (disabled)
// fbROPPDrag(
//     bEnable := bROPPDragEnable,
//     bEStop := IbEmergencyStop,
//     bRun := VIS_ROPP.bROPPDragRun,
//     bPrepare := bROPPDragPrepareRun,
//     bHoming := bROPPDragDoHoming,
//     bHomingDirection := TRUE,
//     bHeightSet := bROPPDragHeightSet,
//     bIgnoreError := VIS_ROPP.bROPPDragIgnoreError,
//     bReset := ROPPDragError.bReset,
//     bResetCycle := P00_PackML.rtCycleReseting.Q,
//     lrMinPosition := 0,
//     lrMaxPosition := 135,
//     lrStartPosition := 3,
//     lrMiddlePosition := 134,
//     lrEndPosition := 134,
//     lrLeadActuatorMoveUpPosition := 15,
//     lrDragAcceleration := 1400,
//     lrDragDeceleration := 1400,
//     lrDragJerk := 25000,
//     lrDragSpeed := lrROPPDragVelocity,
//     bHomingSensor := IbROPPDragHomingSensor,
//     bDragUpSensor := IbROPPDragUpSensor,
//     bDragDownSensor := IbROPPDragDownSensor,
//     bLead1UpSensor := IbROPPDragLeadBefore1UpSensor AND IbROPPDragLeadBefore2UpSensor,
//     bLead2UpSensor := fbROPPDrag.bLeadBefore2Actuator,
//     bManualMovement := bManualMode,
//     iStationIndex := 70,
//     wsStationName := "Przeciąganie formatek ROPP",
//     bManualDragActuator := VIS_ROPP.bROPPDragManualFork,
//     bManualLeadBefore1Actuator := VIS_ROPP.bROPPDragManualLead,
//     bManualLeadBefore2Actuator := bTemp,
//     bManualDragRight := VIS_ROPP.bROPPDragManualRight,
//     bManualDragLeft := VIS_ROPP.bROPPDragManualLeft,
//     DragAxisRef := aROPPDragAxisRef,
//     eRunningState => eROPPDragRunningState,
//     bError => ROPPDragError.bError,
//     udiErrorID => ROPPDragError.nErrorCode,
//     sErrorDescription => ROPPDragError.sErrorString,
//     sErrorDescription2 => ROPPDragError.sErrorString2,
//     sErrorStationName => ROPPDragError.sStationName,
//     udiStationID => ROPPDragError.udiStationID,
//     bDragActuator => QbROPPDragActuator,
//     bLeadBefore1Actuator => QbROPPDragLeadBefore1Actuator,
//     lrActualDragPosition => VIS_ROPP.lrROPPDragPositionCV); // FB_FormsDragStepper
// eROPPDragState := fbROPPDrag.eState;
END_ACTION

ACTION a6_Capping:
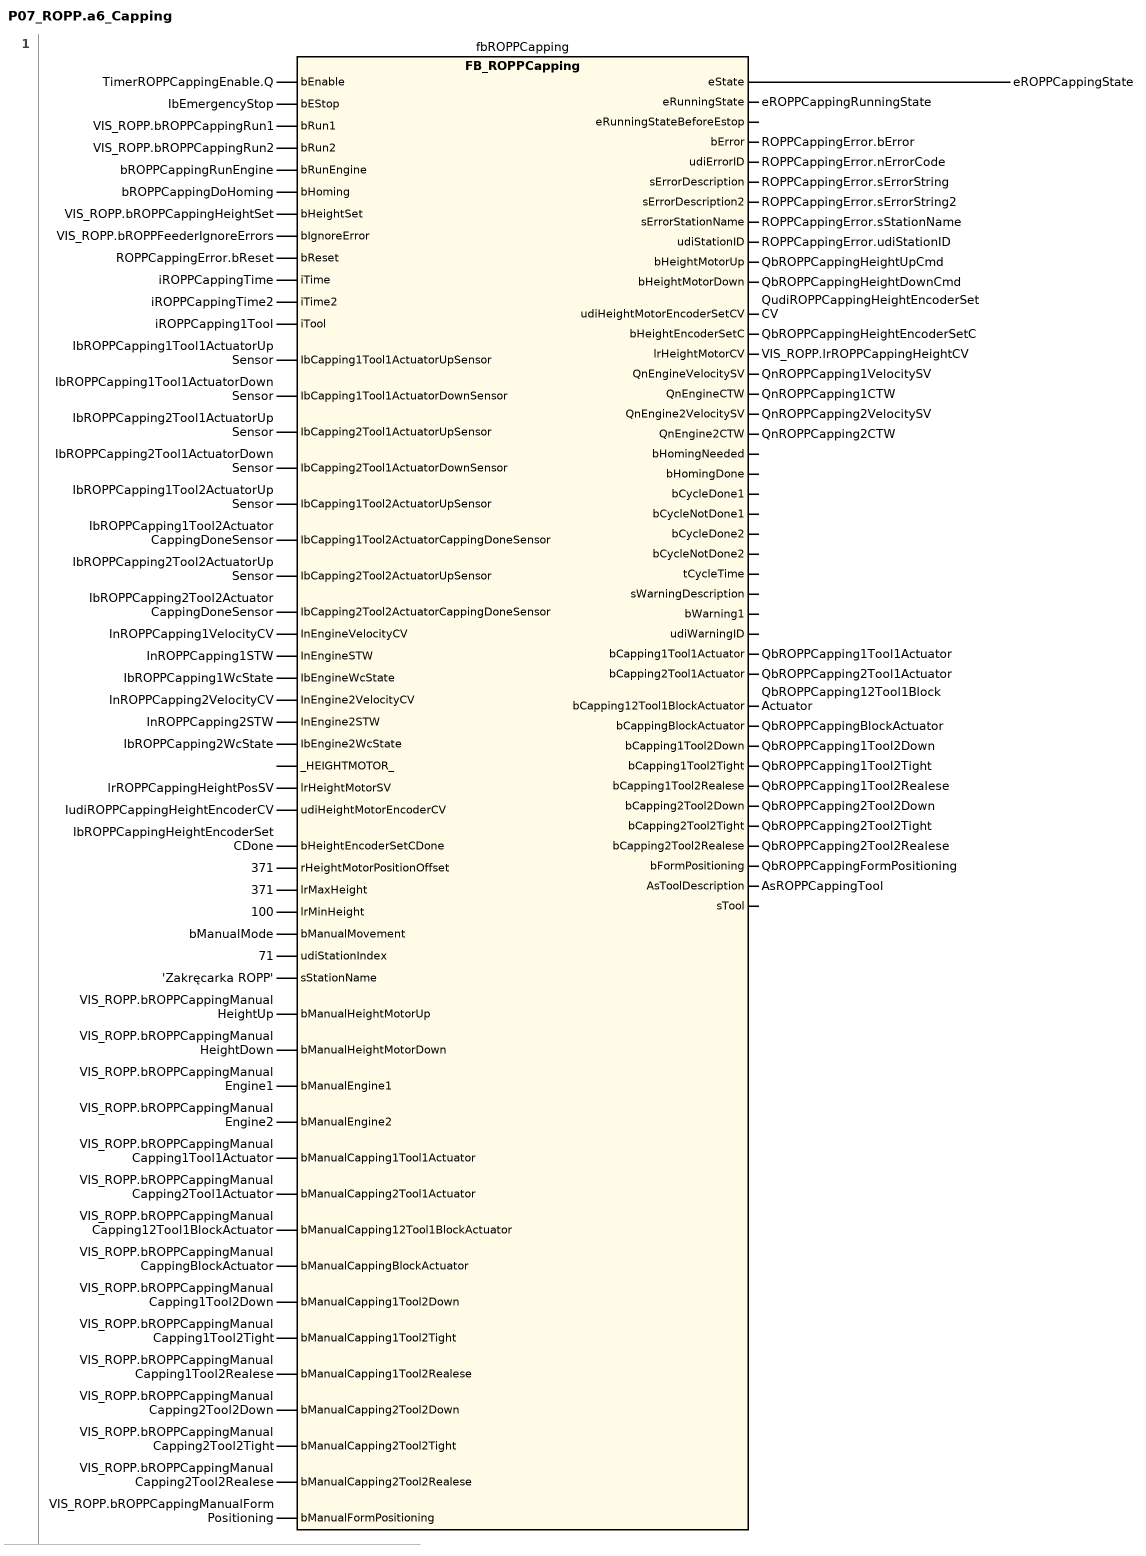
// NETWORK 1
fbROPPCapping(
    bEnable := TimerROPPCappingEnable.Q,
    bEStop := IbEmergencyStop,
    bRun1 := VIS_ROPP.bROPPCappingRun1,
    bRun2 := VIS_ROPP.bROPPCappingRun2,
    bRunEngine := bROPPCappingRunEngine,
    bHoming := bROPPCappingDoHoming,
    bHeightSet := VIS_ROPP.bROPPCappingHeightSet,
    bIgnoreError := VIS_ROPP.bROPPFeederIgnoreErrors,
    bReset := ROPPCappingError.bReset,
    iTime := iROPPCappingTime,
    iTime2 := iROPPCappingTime2,
    iTool := iROPPCapping1Tool,
    IbCapping1Tool1ActuatorUpSensor := IbROPPCapping1Tool1ActuatorUpSensor,
    IbCapping1Tool1ActuatorDownSensor := IbROPPCapping1Tool1ActuatorDownSensor,
    IbCapping2Tool1ActuatorUpSensor := IbROPPCapping2Tool1ActuatorUpSensor,
    IbCapping2Tool1ActuatorDownSensor := IbROPPCapping2Tool1ActuatorDownSensor,
    IbCapping1Tool2ActuatorUpSensor := IbROPPCapping1Tool2ActuatorUpSensor,
    IbCapping1Tool2ActuatorCappingDoneSensor := IbROPPCapping1Tool2ActuatorCappingDoneSensor,
    IbCapping2Tool2ActuatorUpSensor := IbROPPCapping2Tool2ActuatorUpSensor,
    IbCapping2Tool2ActuatorCappingDoneSensor := IbROPPCapping2Tool2ActuatorCappingDoneSensor,
    InEngineVelocityCV := InROPPCapping1VelocityCV,
    InEngineSTW := InROPPCapping1STW,
    IbEngineWcState := IbROPPCapping1WcState,
    InEngine2VelocityCV := InROPPCapping2VelocityCV,
    InEngine2STW := InROPPCapping2STW,
    IbEngine2WcState := IbROPPCapping2WcState,
    lrHeightMotorSV := lrROPPCappingHeightPosSV,
    udiHeightMotorEncoderCV := IudiROPPCappingHeightEncoderCV,
    bHeightEncoderSetCDone := IbROPPCappingHeightEncoderSetCDone,
    rHeightMotorPositionOffset := 371,
    lrMaxHeight := 371,
    lrMinHeight := 100,
    bManualMovement := bManualMode,
    udiStationIndex := 71,
    sStationName := 'Zakręcarka ROPP',
    bManualHeightMotorUp := VIS_ROPP.bROPPCappingManualHeightUp,
    bManualHeightMotorDown := VIS_ROPP.bROPPCappingManualHeightDown,
    bManualEngine1 := VIS_ROPP.bROPPCappingManualEngine1,
    bManualEngine2 := VIS_ROPP.bROPPCappingManualEngine2,
    bManualCapping1Tool1Actuator := VIS_ROPP.bROPPCappingManualCapping1Tool1Actuator,
    bManualCapping2Tool1Actuator := VIS_ROPP.bROPPCappingManualCapping2Tool1Actuator,
    bManualCapping12Tool1BlockActuator := VIS_ROPP.bROPPCappingManualCapping12Tool1BlockActuator,
    bManualCappingBlockActuator := VIS_ROPP.bROPPCappingManualCappingBlockActuator,
    bManualCapping1Tool2Down := VIS_ROPP.bROPPCappingManualCapping1Tool2Down,
    bManualCapping1Tool2Tight := VIS_ROPP.bROPPCappingManualCapping1Tool2Tight,
    bManualCapping1Tool2Realese := VIS_ROPP.bROPPCappingManualCapping1Tool2Realese,
    bManualCapping2Tool2Down := VIS_ROPP.bROPPCappingManualCapping2Tool2Down,
    bManualCapping2Tool2Tight := VIS_ROPP.bROPPCappingManualCapping2Tool2Tight,
    bManualCapping2Tool2Realese := VIS_ROPP.bROPPCappingManualCapping2Tool2Realese,
    bManualFormPositioning := VIS_ROPP.bROPPCappingManualFormPositioning,
    eRunningState => eROPPCappingRunningState,
    bError => ROPPCappingError.bError,
    udiErrorID => ROPPCappingError.nErrorCode,
    sErrorDescription => ROPPCappingError.sErrorString,
    sErrorDescription2 => ROPPCappingError.sErrorString2,
    sErrorStationName => ROPPCappingError.sStationName,
    udiStationID => ROPPCappingError.udiStationID,
    bHeightMotorUp => QbROPPCappingHeightUpCmd,
    bHeightMotorDown => QbROPPCappingHeightDownCmd,
    udiHeightMotorEncoderSetCV => QudiROPPCappingHeightEncoderSetCV,
    bHeightEncoderSetC => QbROPPCappingHeightEncoderSetC,
    lrHeightMotorCV => VIS_ROPP.lrROPPCappingHeightCV,
    QnEngineVelocitySV => QnROPPCapping1VelocitySV,
    QnEngineCTW => QnROPPCapping1CTW,
    QnEngine2VelocitySV => QnROPPCapping2VelocitySV,
    QnEngine2CTW => QnROPPCapping2CTW,
    bCapping1Tool1Actuator => QbROPPCapping1Tool1Actuator,
    bCapping2Tool1Actuator => QbROPPCapping2Tool1Actuator,
    bCapping12Tool1BlockActuator => QbROPPCapping12Tool1BlockActuator,
    bCappingBlockActuator => QbROPPCappingBlockActuator,
    bCapping1Tool2Down => QbROPPCapping1Tool2Down,
    bCapping1Tool2Tight => QbROPPCapping1Tool2Tight,
    bCapping1Tool2Realese => QbROPPCapping1Tool2Realese,
    bCapping2Tool2Down => QbROPPCapping2Tool2Down,
    bCapping2Tool2Tight => QbROPPCapping2Tool2Tight,
    bCapping2Tool2Realese => QbROPPCapping2Tool2Realese,
    bFormPositioning => QbROPPCappingFormPositioning,
    AsToolDescription => AsROPPCappingTool); // FB_ROPPCapping
eROPPCappingState := fbROPPCapping.eState;
END_ACTION

ACTION a7_CappingCheck:

fbIbROPPCappingCheckSensor(bIN:= IbROPPCappingCheckSensor, tFilterTimeOn:=T#0MS , tFilterTimeOff:= T#0MS, bOUT=> );
fbIbROPPCappingCheckSensor.bOUT;

//Wizka
VIS_ROPP.bROPPCappingCheckOK	:=	fbIbROPPCappingCheckSensor.bOUT;
END_ACTION

ACTION aButtons:
//Dodane
IbROPPCycleStartButton;
//IbSafetyResetIn;
IbROPPCycleStopButton;
END_ACTION

ACTION aLimits:
(*
Nazwa:			aLimits
Opis:			Zabezpieczenia
Wersja:			v1.0
Data:			2023-11-24
Autor:			DP
Urzadzenia:		
Zmiany:	

Info:
*)

(**** Limity i zabezpieczenia***)
IF lrROPPDragVelocity <50 THEN	lrROPPDragVelocity	:= 50;	END_IF 

IF 	VIS.lrROPPDragStationStartPosition		= 0		THEN	VIS.lrROPPDragStationStartPosition		:=	3;		END_IF;
IF 	VIS.lrROPPDragStationEndPosition		= 0		THEN	VIS.lrROPPDragStationEndPosition		:=	134;	END_IF;
END_ACTION

ACTION aPneumatics:
// Do podpięcia według kolejności

//N8 - GÓRA
QbROPPCapping1Tool1Actuator; //gora dol  zakrecarka M1
QbROPPCapping2Tool1Actuator; //gora dol  zakrecarka M2
QbROPPCapping12Tool1BlockActuator;
QbROPPCappingBlockActuator;
QbROPPCapping1Tool2Down;		
QbROPPCapping1Tool2Tight;		
QbROPPCapping2Tool2Down;		
QbROPPCapping2Tool2Tight;	
//N8A - DÓŁ
QbROPPDragActuator;	// widly gora dol
QbROPPDragLeadBefore1Actuator;		//prowadnice 52N8.1A/B2, 52N8.1A/B3
QbROPPStoperBeforeActuator; //silownik horyzontalny N8A
QbROPPCappingFormPositioning;//indeksowanie formatek
QbROPPStoperAfterActuator; //silownik horyzontalny N8A
//Rezerwa
//Rezerwa
(*************************** ROPP EB1 **************************************)
// Wyspa 1 - dozowanie
IuiPneumaticROPPEB1State;
QABPneumaticROPPEB1ValveCoils[1].0	:= QbROPPCapping1Tool1Actuator;			//[810, 5/3, podnoszenie stacji 1]
QABPneumaticROPPEB1ValveCoils[1].1 	:= FALSE;                                               
QABPneumaticROPPEB1ValveCoils[1].2 	:= QbROPPCapping2Tool1Actuator; 		//[820, 5/3, podnoszenie stacji 2]
QABPneumaticROPPEB1ValveCoils[1].3 	:= FALSE;                        	                    
QABPneumaticROPPEB1ValveCoils[1].4 	:= QbROPPCappingBlockActuator;			
QABPneumaticROPPEB1ValveCoils[1].5 	:= QbROPPCapping12Tool1BlockActuator;                                              
QABPneumaticROPPEB1ValveCoils[1].6 	:= QbROPPCapping1Tool2Down;; 			
QABPneumaticROPPEB1ValveCoils[1].7 	:= NOT QbROPPCapping1Tool2Down;//QbROPPCapping1Tool2Tight;                                            
QABPneumaticROPPEB1ValveCoils[2].0 	:= NOT QbROPPCapping1Tool2Tight;//QbROPPCapping1Tool2Realese;//QbROPPCapping1Tool2Tight;//FALSE;				
QABPneumaticROPPEB1ValveCoils[2].1  := QbROPPCapping1Tool2Tight;                                                      
QABPneumaticROPPEB1ValveCoils[2].2 	:= QbROPPCapping2Tool2Down;; 	
QABPneumaticROPPEB1ValveCoils[2].3 	:= NOT QbROPPCapping2Tool2Down;//QbROPPCapping2Tool2Tight;  
QABPneumaticROPPEB1ValveCoils[2].4 	:= NOT QbROPPCapping2Tool2Tight;//QbROPPCapping2Tool2Realese;//QbROPPCapping2Tool2Tight;//FALSE;											
QABPneumaticROPPEB1ValveCoils[2].5 	:= QbROPPCapping2Tool2Tight;                              
QABPneumaticROPPEB1ValveCoils[2].6 	:= QbROPPDragActuator;                               
QABPneumaticROPPEB1ValveCoils[2].7 	:= NOT QbROPPDragActuator;
QABPneumaticROPPEB1ValveCoils[3].0 	:= QbROPPDragLeadBefore1Actuator;
QABPneumaticROPPEB1ValveCoils[3].1  := NOT QbROPPDragLeadBefore1Actuator;                                                   
QABPneumaticROPPEB1ValveCoils[3].2 	:= QbROPPStoperBeforeActuator;	                                //[8A20, 5/3, podnoszenie stacji 2]
QABPneumaticROPPEB1ValveCoils[3].3  := FALSE;                                                      
QABPneumaticROPPEB1ValveCoils[3].4 	:= QbROPPCappingFormPositioning;	                                //[8A30, 5/2, głowica 1 ruch góra-dół, indeksowanie formatek]
QABPneumaticROPPEB1ValveCoils[3].5  := FALSE;                                                       
QABPneumaticROPPEB1ValveCoils[3].6 	:= QbROPPStoperAfterActuator;                               //[8A40, 5/2, głowica 2 ruch góra-dół]	
QABPneumaticROPPEB1ValveCoils[3].7  := FALSE;                                                 
QABPneumaticROPPEB1ValveCoils[4].0 	;		                                
QABPneumaticROPPEB1ValveCoils[4].1  ;                                       
QABPneumaticROPPEB1ValveCoils[4].2 	;		                                
QABPneumaticROPPEB1ValveCoils[4].3  ;                                      
QABPneumaticROPPEB1ValveCoils[4].4 	;		                                
QABPneumaticROPPEB1ValveCoils[4].5  ;        
QABPneumaticROPPEB1ValveCoils[4].6 	;		
QABPneumaticROPPEB1ValveCoils[4].7  ; 
                                                               
(*********************Koniec ROPP EB1 **************************************) 


//Zawór głównego powietrza
QbROPPCompressedAir	:=	IbEmergencyStop;

(*************************** EB1 **************************************)
// Wyspa 1 - 52N8
IuiPneumaticROPPEB1State;
//DI1
IbROPPCapping1Tool1ActuatorDownSensor		 					:=	IABPneumaticROPPEB1DigitalInput[1].0;	
IbROPPCapping1Tool1ActuatorUpSensor						:=	IABPneumaticROPPEB1DigitalInput[1].1;	
IbROPPCapping2Tool1ActuatorDownSensor		 					:=	IABPneumaticROPPEB1DigitalInput[1].2;	
IbROPPCapping2Tool1ActuatorUpSensor						:=	IABPneumaticROPPEB1DigitalInput[1].3;
IbROPPPuttedCheckSensor										:=	IABPneumaticROPPEB1DigitalInput[1].4;	//52N8W5 obecnosc metalowego korka na butli przed zakreceniem nad pierwszym RFID
IbROPPCappingCheckSensor									:=	IABPneumaticROPPEB1DigitalInput[1].5;		//52N8W6 obecnosc metalowego korka na butli po zakreceniu
IbROPPFeederAirOK											:=	IABPneumaticROPPEB1DigitalInput[1].6;		
IbROPPFeederCapsWheelLevel									:=	IABPneumaticROPPEB1DigitalInput[1].7;	//52N8W8 czujnik zapelnienia bebna, flaga na dnie bebna
//DI2                                               		
IbROPPFeederCapsLevel										:=	IABPneumaticROPPEB1DigitalInput[2].0;	// 52N8.2/B9 poziom kapsli w bebnie
IbROPPFeederCapsSleeveUp (*odwrotny*)						:=	NOT IABPneumaticROPPEB1DigitalInput[2].1;	//52N8.2/B10 nakretka w rekawie wyzej
															;	IABPneumaticROPPEB1DigitalInput[2].2;	//52N8.2/B11 nakretka w rekawie nizej. brak czujnika 17.02.2025 pewnie wypadnie z projektu
IbROPPCapping1Tool2ActuatorUpSensor							:=	IABPneumaticROPPEB1DigitalInput[2].3;	
IbROPPCapping1Tool2ActuatorCappingDoneSensor				:=	IABPneumaticROPPEB1DigitalInput[2].4;	
IbROPPCapping2Tool2ActuatorCappingDoneSensor				:=	IABPneumaticROPPEB1DigitalInput[2].5;		
IbROPPCapping2Tool2ActuatorUpSensor							:=	IABPneumaticROPPEB1DigitalInput[2].6;		
																IABPneumaticROPPEB1DigitalInput[2].7;	

// Wyspa 1 - 52N8A
IuiPneumaticROPPEB1State;
//DI1
IbROPPDragHomingSensor					 					:=	IABPneumaticROPPEB1DigitalInput[3].0;	
IbROPPDragLeadBefore1UpSensor								:=	IABPneumaticROPPEB1DigitalInput[3].1;	
IbROPPDragLeadBefore2UpSensor		 						:=	IABPneumaticROPPEB1DigitalInput[3].2;	
IbROPPDragUpSensor											:=	IABPneumaticROPPEB1DigitalInput[3].3;
IbROPPDragDownSensor										:=	IABPneumaticROPPEB1DigitalInput[3].4;	
IbROPPCappingFormPositioningOnSensor						:=	IABPneumaticROPPEB1DigitalInput[3].5;		
IbROPPCappingFormPositioningOffSensor						:=	IABPneumaticROPPEB1DigitalInput[3].6;		
IbROPPThirdFormSensor 										:=	IABPneumaticROPPEB1DigitalInput[3].7;	//52N8.1A/B8  obecnosc formatki pod zakrecarka
//DI2                                               		
IbROPPBeforeSevenFormSensor									:=	IABPneumaticROPPEB1DigitalInput[4].0;
(*IbROPPCappingCheckFormSensor								:=*)IABPneumaticROPPEB1DigitalInput[4].0;	//52N8.2A/B9 druga glowica RFID
IbROPPSevenFormSensor										:=	IABPneumaticROPPEB1DigitalInput[4].1;	//52N8.2A/B10 sprawdzanie obecnosci formatki przy pierwszej glowicy RFID
IbROPPAfterFormSensor										:=	IABPneumaticROPPEB1DigitalInput[4].2;	//Najbliżej ROPP	
IbROPPAfter2FormSensor										:=	IABPneumaticROPPEB1DigitalInput[4].3;	//Dalej ROPP (Na ukos)
IbROPPAfter3FormSensor										:=	IABPneumaticROPPEB1DigitalInput[4].4;	//Najdalej ROPP 
																IABPneumaticROPPEB1DigitalInput[4].5;		
																IABPneumaticROPPEB1DigitalInput[4].6;		
																IABPneumaticROPPEB1DigitalInput[4].7;	
(*********************Koniec EB2 **************************************)
END_ACTION

ACTION aPowerSupply:


	//Dodane do głwnych
	IbROPPFuseFB1OK	; //BC6 Blok bezpiecznikowy	
	IbROPPFuseFB2OK	; //BC6 Zasilanie safety
	IbROPPFuseFB3OK	; //Glowica 1	
	IbROPPFuseFB4OK	; //Glowica 2
	IbROPPFuseFB5OK	; //Koło podajnika
	IbROPPFuseFB6OK	; //Spowalniacz
	IbROPPFuseFB7OK	; //Transporter za stacją
	IbROPPFuseFB8OK	; //Podnośnik podajnika
	IbROPPFuseFB9OK	; //Podnośnik zakrecarek
END_ACTION

ACTION aRFID:
(*Przepisanie bity wykrycia karty*)
bReadedCardBeforeROPP 		:= IbBeforeROPPReaderTagPresent AND fbBeforeROPPReader.bCodeReaded;
nReadedCardBeforeROPP 		:= DINT_TO_ULINT(fbBeforeROPPReader.diReadedCode);

bReadedCardAfterROPP 		:= IbAfterROPPReaderTagPresent AND fbAfterROPPReader.bCodeReaded;
nReadedCardAfterROPP 		:= DINT_TO_ULINT(fbAfterROPPReader.diReadedCode);
END_ACTION

ACTION aRFID_FB:
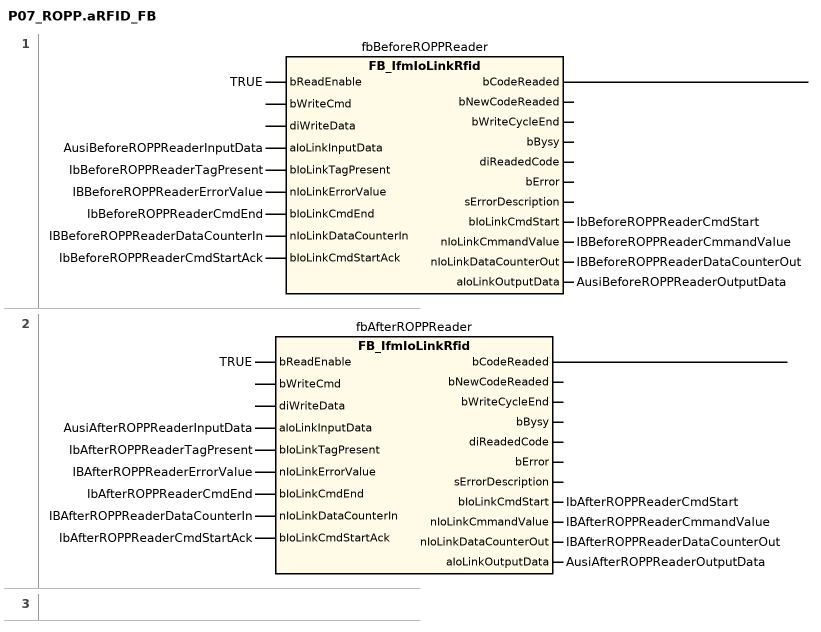
// NETWORK 1
fbBeforeROPPReader(
    bReadEnable := TRUE,
    aIoLinkInputData := AusiBeforeROPPReaderInputData,
    bIoLinkTagPresent := IbBeforeROPPReaderTagPresent,
    nIoLinkErrorValue := IBBeforeROPPReaderErrorValue,
    bIoLinkCmdEnd := IbBeforeROPPReaderCmdEnd,
    nIoLinkDataCounterIn := IBBeforeROPPReaderDataCounterIn,
    bIoLinkCmdStartAck := IbBeforeROPPReaderCmdStartAck,
    bIoLinkCmdStart => IbBeforeROPPReaderCmdStart,
    nIoLinkCmmandValue => IBBeforeROPPReaderCmmandValue,
    nIoLinkDataCounterOut => IBBeforeROPPReaderDataCounterOut,
    aIoLinkOutputData => AusiBeforeROPPReaderOutputData); // FB_IfmIoLinkRfid

// NETWORK 2
fbAfterROPPReader(
    bReadEnable := TRUE,
    aIoLinkInputData := AusiAfterROPPReaderInputData,
    bIoLinkTagPresent := IbAfterROPPReaderTagPresent,
    nIoLinkErrorValue := IBAfterROPPReaderErrorValue,
    bIoLinkCmdEnd := IbAfterROPPReaderCmdEnd,
    nIoLinkDataCounterIn := IBAfterROPPReaderDataCounterIn,
    bIoLinkCmdStartAck := IbAfterROPPReaderCmdStartAck,
    bIoLinkCmdStart => IbAfterROPPReaderCmdStart,
    nIoLinkCmmandValue => IBAfterROPPReaderCmmandValue,
    nIoLinkDataCounterOut => IBAfterROPPReaderDataCounterOut,
    aIoLinkOutputData => AusiAfterROPPReaderOutputData); // FB_IfmIoLinkRfid

// NETWORK 3
END_ACTION

ACTION aSafety:

// Dodać do P00_Alarms.aGeneralAlarms
	IbROPPEmergencyStopButton0Pressed;
	IbROPPEmergencyStopButton1Pressed;
	
(*
	IF IbROPPEmergencyStopButton0Pressed THEN
		GeneralAlarms.nErrorCode:=1;			
		GeneralAlarms.sErrorString:='Stop Awaryjny, sprawdź bezpieczeństwo, zresetuj przyciskiem na panelu | Naciśnięty przycisk awaryjny 1 na ROPP';	
	ELSIF  IbROPPEmergencyStopButton1Pressed THEN
		GeneralAlarms.nErrorCode:=2;
		GeneralAlarms.sErrorString:='Stop Awaryjny, sprawdź bezpieczeństwo, zresetuj przyciskiem na panelu | Naciśnięty przycisk awaryjny 2 na ROPP';	
*)	
	

// Dodać do miejsca gdzie są zamykane drzwi	
// lub zostawić tak jak jest
	QbROPPDoors0Close := QbDispencersDoorsClose;
    QbROPPDoors1Close := QbDispencersDoorsClose;
END_ACTION

ACTION aSignalization:
(*****Listwy LED*****)

QiROPPRedSignalizationLamp		:= P00_Signalization.QiLineRedSignalizationLamp;
QiROPPGreenSignalizationLamp	:= P00_Signalization.QiLineGreenSignalizationLamp;
QiROPPBlueSignalizationLamp		:= P00_Signalization.QiLineBlueSignalizationLamp;
QiROPPWhiteSignalizationLamp	:= P00_Signalization.QiLineWhiteSignalizationLamp;

QbROPPStartLamp	:= P00_Signalization.QbStartLamp;	   
QbROPPResetLamp	:= P00_Signalization.QbResetLamp;
END_ACTION

ACTION aWarnings:

END_ACTION

END_PROGRAM

// ---- POUs/FB/FB_MitsubishiInverter.TcPOU
FUNCTION_BLOCK FB_MitsubishiInverter
VAR_INPUT
	bEnable												: BOOL;					// Uruchomienie bloku
	bWcState											: BOOL;
	bEStop												: BOOL;					// Pozwolenie na prace bloku z SAFETY (TRUE-maszyna gotowa do pracy FALSE-brak pozolenia na prace)
	bExternalError										: BOOL;
	bRun												: BOOL;					// Komenda na uruchomienie 
	bDirection											: BOOL;					// Kierunek obrotow silnika 
	bReset												: BOOL;					// Reset falownika po bledzie
	bManualMode											: BOOL;					// Tryb manualny
	bJogForward											: BOOL;					// Komenda na ruch w kierunku dodatnim
	bJogBackward										: BOOL;					// Komenda na ruch w kierunku ujemnym 
	sStationName										: WSTRING(200);
	iStationIndex										: UDINT;
	udiSetVelocity										: UDINT;
	udiActualVelocity				(*AT %Q**)			: UDINT;
	uiStatusWord					(*AT %Q**)			: UINT;			//
	uiErrorCode											: UINT;
END_VAR
VAR_OUTPUT
	eState												: E_Station;			// Stan pracy bloku
	eRunningState										: E_ConveyorState;
	bError												: BOOL;					// Blad falownika
	udiErrorID											: UDINT;				// Nr błędu bloku funkcyjnego
	sErrorDescription									: STRING(200);			// Opis błędu
	sErrorDescription2									: STRING(200);			// Opis błędu
	udiStationID										: UDINT;				// Nr stacji	
	sErrorStationName									: STRING;				// Nazwa stacji
	uiControlWord					(*AT %I**)			: UINT;
	udiTargetVelocity				(*AT %I**)			: UDINT;
END_VAR
VAR
	rtRun												: R_TRIG;	
	
	tonCheckInitTime									: TON;
	tonRessetingState									: TON;
	
	iPreparingToReadyStep								: INT;
	//ControlWord
	bSwitchOn											: BOOL;
	bEnableVoltage										: BOOL;
	bQuickStop											: BOOL;
	bFaultReset											: BOOL;
	bEnableOperation									: BOOL;
	
	//StatusWord
	bReadyToSwitchOn									: BOOL;
	bSwitchedOn											: BOOL;
	bOperationEnabled									: BOOL;
	bFault												: BOOL;
	bQuickStopStatus									: BOOL;
	bSwitchOnDisabled									: BOOL;
	bWarning											: BOOL;
	bRemote												: BOOL;
	bInternalLimitActive								: BOOL;
	
	//Errors
	bCheckInitTimeError									: BOOL;
	bWcStateError										: BOOL;
	bMitsubishiReadinessError							: BOOL;
	
	tonbSwitchedOn: TON;
	
	//Zmienne od EVENTLOGGER
	bAlarmInit 						: BOOL := TRUE; 
	nAlarmNumerator					: INT;
	arfbAlarm						: ARRAY[0..19] OF  FB_TcAlarm;		//Tablica bloczków błędów
	fbSourceInfo 					: FB_TcSourceInfo;
	iSourceInfo						: I_TcSourceInfo;
	sAlarmTest						: STRING;
	//Koniec zmiennych od EVENTLOGGER
END_VAR

aStationID();
ACT_Signals();
ACT_EStop();						
ACT_ErrorHandling();


IF NOT bEnable THEN
	IF eState <> E_Station.eDisabled AND eState <> E_Station.ePreparingToDisable THEN //Nie mogę wyłączyć falownik podczas awaryjnego zatrzymania (STO)
		eState					:= E_Station.ePreparingToDisable;
		eRunningState			:= E_ConveyorState.ePreparingToDisable;
	END_IF
END_IF


CASE eState OF
	
	E_Station.eDisabled: 			// Stan nieaktywnosci (Stacja wyłączona)
		
		State_Disabled();
	
		
	E_Station.eAborted: 			// Stan bezpiecznego zatrzymania (po Abortingu) 
	
		State_Aborted();
		
	
	E_Station.eAborting:			// Stan bezpiecznego zatrzymywania (po EStopie) 
	
		State_Aborting();
		
	
	E_Station.eError:				// Stan błędu 
	
		State_Error();
	
		
	E_Station.eResetting:			// Stan resetowania bledu (po Errorze)
	
		State_Resetting();
		
	
	E_Station.eManualMovement:		// Stan ruchów manualnych 
	
		State_ManualMovement();
		
	
	E_Station.eHoming:				// Stan bazowania 
	
		State_Homing();
		
	
	E_Station.eHomingDone:			// Stan wykonania bazowania
	
		State_HomingDone();
		
	
	E_Station.ePreparingToReady:	// Stan przygotowywania do gotowosci (zawsze przed Ready)
	
		State_PreparingToReady();
		
	
	E_Station.ePreparingToDisable:	// Stan przygotowywania do nieaktywnosci (po wyłączeniu Enable)
	
		State_PreparingToDisable();
	
		
	E_Station.eReady:				// Stan gotowosci
	
		State_Ready();
		
	
	E_Station.eStopping:			// Stan zatrzymywania 
	
		State_Stopping();
		
		
	E_Station.eStarting:			// Stan uruchamiania (po Ready)
	
		State_Starting();
			
	
	E_Station.eRunning:				// Stan wykonywania cyklu (po Startingu), w tym stanie osobny
	
		State_Running();

END_CASE

ACTION ACT_ErrorHandling:
// Alarm_0180	180	Error	Błąd Falownika {0}
// Alarm_0181	181	Error	Przekroczenie czasu oczekiwania na odpowiedź falownika
// Alarm_0182	182	Error	Błąd komunikacji z urządzeniem (WcState)
// Alarm_0183	183	Error	Utracono gotowość falownika do pracy
// Alarm_0184	184	Error	Sprawdź zabezpieczenie silnikowe

IF bAlarmInit THEN
    bAlarmInit := FALSE; 
	fbSourceInfo.Clear();
	fbSourceInfo.sName:=wsLiteral_TO_UTF8(sStationName);//'Machine';
	fbSourceInfo.nId:=udiStationID;//2700;
	// Alarm_0180	180	Error	Błąd Falownika
    arfbAlarm[0].CreateEx(stEventEntry := TC_EVENTS.AlarmClass.Alarm_0180, bWithConfirmation:= FALSE,  ipSourceInfo:= fbSourceInfo); 
	// Alarm_0181	181	Error	Przekroczenie czasu oczekiwania na odpowiedź falownika
	arfbAlarm[1].CreateEx(stEventEntry := TC_EVENTS.AlarmClass.Alarm_0181, bWithConfirmation:= FALSE,  ipSourceInfo:= fbSourceInfo);
	// Alarm_0182	182	Error	Błąd komunikacji z urządzeniem (WcState)
	arfbAlarm[2].CreateEx(stEventEntry := TC_EVENTS.AlarmClass.Alarm_0182, bWithConfirmation:= FALSE,  ipSourceInfo:= fbSourceInfo); 
	// Alarm_0183	183	Error	Utracono gotowość falownika do pracy
	arfbAlarm[3].CreateEx(stEventEntry := TC_EVENTS.AlarmClass.Alarm_0183, bWithConfirmation:= FALSE,  ipSourceInfo:= fbSourceInfo); 
	// Alarm_0184	184	Error	Sprawdź zabezpieczenie silnikowe
	arfbAlarm[4].CreateEx(stEventEntry := TC_EVENTS.AlarmClass.Alarm_0184, bWithConfirmation:= FALSE,  ipSourceInfo:= fbSourceInfo); 
END_IF








tonCheckInitTime.IN								:= eState = E_Station.ePreparingToReady OR eState = E_Station.eStarting OR eState = E_Station.eStopping;
tonCheckInitTime.PT								:= T#10S;
tonCheckInitTime();

IF tonCheckInitTime.Q  THEN
	bCheckInitTimeError							:= TRUE;
END_IF

IF bWcState THEN
	bWcStateError								:= TRUE;
END_IF

//IF NOT bSwitchedOn THEN
IF	tonbSwitchedOn.Q THEN
	IF eState = E_Station.eReady OR eState = E_Station.eStarting OR eState = E_Station.eRunning OR
	   eState = E_Station.eStopping OR eState = E_Station.eManualMovement THEN
	   
	   bMitsubishiReadinessError				:= TRUE;
	END_IF
END_IF

//bError											:= bFault OR bCheckInitTimeError OR bWcStateError OR bMitsubishiReadinessError OR bExternalError;

// Alarm_0180	180	Error	Błąd Falownika {0}
IF bFault THEN
	 arfbAlarm[0].ipArguments.Clear() .AddUDInt(uiErrorCode);
	 IF NOT arfbAlarm[0].bActive THEN
			arfbAlarm[0].Raise(nTimeStamp:=0);
		END_IF
	ELSE	
		IF  arfbAlarm[0].bActive AND bReset THEN
			arfbAlarm[0].Clear(nTimeStamp:=0, bResetConfirmation:= FALSE);
		END_IF	
// 	udiErrorID									:= 121;
// //	udiErrorID									:= uiErrorCode;
// 	sErrorDescription							:= 'Błąd Falownika';
// 	sErrorDescription2							:= UINT_TO_STRING(uiErrorCode);
END_IF
// Alarm_0181	181	Error	Przekroczenie czasu oczekiwania na odpowiedź falownika
IF bCheckInitTimeError AND bEnable THEN
	IF NOT arfbAlarm[1].bActive THEN
			arfbAlarm[1].Raise(nTimeStamp:=0);
		END_IF
	ELSE	
		IF  arfbAlarm[1].bActive AND bReset THEN
			arfbAlarm[1].Clear(nTimeStamp:=0, bResetConfirmation:= FALSE);
		END_IF	
// 	udiErrorID									:= 122;
// //	udiErrorID									:= iStationIndex + 1;
// 	sErrorDescription							:= 'Przekroczenie czasu oczekiwania na odpowiedź falownika';
END_IF
// Alarm_0182	182	Error	Błąd komunikacji z urządzeniem (WcState)
IF bWcStateError THEN
		IF NOT arfbAlarm[2].bActive THEN
			arfbAlarm[2].Raise(nTimeStamp:=0);
		END_IF
	ELSE	
		IF  arfbAlarm[2].bActive AND bReset THEN
			arfbAlarm[2].Clear(nTimeStamp:=0, bResetConfirmation:= FALSE);
		END_IF	
// 	udiErrorID									:= 123;
// // udiErrorID									:= iStationIndex + 2;
// 	sErrorDescription							:= 'Błąd komunikacji z urządzeniem (WcState)';
END_IF
// Alarm_0183	183	Error	Utracono gotowość falownika do pracy
IF bMitsubishiReadinessError THEN
		IF NOT arfbAlarm[3].bActive THEN
			arfbAlarm[3].Raise(nTimeStamp:=0);
		END_IF
	ELSE	
		IF  arfbAlarm[3].bActive AND bReset THEN
			arfbAlarm[3].Clear(nTimeStamp:=0, bResetConfirmation:= FALSE);
		END_IF	
// 	udiErrorID									:= 124;
// //	udiErrorID										:= iStationIndex + 3;
// 	sErrorDescription							:= 'Utracono gotowość falownika do pracy';
END_IF
// Alarm_0184	184	Error	Sprawdź zabezpieczenie silnikowe
IF bExternalError THEN
		IF NOT arfbAlarm[4].bActive THEN
			arfbAlarm[4].Raise(nTimeStamp:=0);
		END_IF
	ELSE	
		IF  arfbAlarm[4].bActive AND bReset THEN
			arfbAlarm[4].Clear(nTimeStamp:=0, bResetConfirmation:= FALSE);
		END_IF	
// 	udiErrorID									:= 125;
// //	udiErrorID									:= iStationIndex + 4;
// 	sErrorDescription							:= 'Sprawdź zabezpieczenie silnikowe';
END_IF


IF NOT bEnable THEN
	bError										:= FALSE;
	udiErrorID									:= 0;
	sErrorDescription							:= '';
	sErrorDescription2							:= '';
END_IF

IF bError THEN
	
	IF eState = E_Station.ePreparingToReady OR eState = E_Station.eReady OR eState = E_Station.eStarting OR
	   eState = E_Station.eRunning OR eState = E_Station.eStopping OR eState = E_Station.eManualMovement THEN
	   
	   eState									:= E_Station.eError;
	   eRunningState							:= E_ConveyorState.eError;
	END_IF
END_IF

IF NOT bError THEN
	udiErrorID									:= 0;
	sErrorDescription							:= '';
	sErrorDescription2							:= '';
END_IF

sErrorStationName								:= WSTRING_TO_STRING(sStationName);


(*Wyświetlanie błedu na wyjściu*)
bError							:= FALSE;
FOR nAlarmNumerator := 0 TO 19 DO
	bError						:= bError OR arfbAlarm[nAlarmNumerator].bActive;
END_FOR
END_ACTION

ACTION ACT_EStop:


IF NOT bEStop THEN
	IF eState <> E_Station.eAborted AND eState <> E_Station.eAborting AND eState <> E_Station.eDisabled THEN
		
		eState					:= E_Station.eAborting;	
		eRunningState			:= E_ConveyorState.eAborting;
	END_IF
END_IF
END_ACTION

ACTION ACT_Signals:

rtRun.CLK									:= bRun;
rtRun();

tonRessetingState.IN						:= eState = E_Station.eResetting;
tonRessetingState.PT						:= T#700MS;
tonRessetingState();
tonbSwitchedOn	(IN:=	NOT bSwitchedOn,	PT:=T#1S);


//ControlWord-------------------------
uiControlWord.0				:= bSwitchOn;
uiControlWord.1				:= bEnableVoltage;
uiControlWord.2				:= bQuickStop;
uiControlWord.3				:= bEnableOperation; 
uiControlWord.7				:= bFaultReset;
//------------------------------------

//StatusWord--------------------------

bReadyToSwitchOn			:= uiStatusWord.0;
bSwitchedOn					:= uiStatusWord.1;
bOperationEnabled			:= uiStatusWord.2;
bFault						:= uiStatusWord.3;
bQuickStopStatus			:= uiStatusWord.5;
bSwitchOnDisabled			:= uiStatusWord.6;
bWarning					:= uiStatusWord.7;
bRemote						:= uiStatusWord.9;
bInternalLimitActive		:= uiStatusWord.11;

IF bDirection THEN
	udiTargetVelocity			:= (SINT_TO_UDINT(-1))*udiSetVelocity;
ELSE 
	udiTargetVelocity			:= udiSetVelocity;
END_IF
END_ACTION

ACTION aStationID:
udiStationID	:=	iStationIndex;
END_ACTION

ACTION State_Aborted:


IF bEStop THEN
	
	IF NOT bError THEN
		eState					:= E_Station.ePreparingToReady;
		eRunningState			:= E_ConveyorState.ePreparingToReady;
	ELSE
		eState					:= E_Station.eError;
		eRunningState			:= E_ConveyorState.eError;
	END_IF
	
	IF NOT bEnable THEN
		eState					:= E_Station.ePreparingToDisable;
		eRunningState			:= E_ConveyorState.ePreparingToDisable;
	END_IF
	
END_IF
// No w KONCU DZIAŁA
END_ACTION

ACTION State_Aborting:

bSwitchOn					:= FALSE;
bEnableVoltage				:= FALSE;
bQuickStop					:= FALSE;
bEnableOperation			:= FALSE;

iPreparingToReadyStep		:= 0;

eState						:= E_Station.eAborted;
eRunningState			:= E_ConveyorState.eAborted;
END_ACTION

ACTION State_Disabled:


IF bEnable THEN
	
	eState					:= E_Station.ePreparingToReady;
	eRunningState			:= E_ConveyorState.ePreparingToReady;
END_IF
END_ACTION

ACTION State_Error:

bSwitchOn				:= FALSE;
bEnableVoltage			:= FALSE;
bQuickStop				:= FALSE;
bEnableOperation		:= FALSE;

iPreparingToReadyStep	:= 0;

IF bReset THEN
	bFaultReset			:= bReset;
	eState				:= E_Station.eResetting;
	eRunningState			:= E_ConveyorState.eResetting;
END_IF
END_ACTION

ACTION State_Homing:

END_ACTION

ACTION State_HomingDone:

END_ACTION

ACTION State_ManualMovement:


IF  bJogForward THEN
	bEnableOperation					:= TRUE;
ELSE
	bEnableOperation					:= FALSE;
	//eState								:= E_Station.eStopping;
END_IF

IF NOT bManualMode THEN
	bEnableOperation					:= FALSE;
	eState								:= E_Station.eStopping;
	eRunningState						:= E_ConveyorState.eStopping;
END_IF
END_ACTION

ACTION State_PreparingToDisable:
bSwitchOn								:= FALSE;
bEnableVoltage							:= FALSE;
bQuickStop								:= FALSE;
bEnableOperation						:= FALSE;
bFaultReset								:= FALSE;

iPreparingToReadyStep					:= 0;

eState									:= E_Station.eDisabled;
eRunningState							:= E_ConveyorState.eDisabled;
END_ACTION

ACTION State_PreparingToReady:


CASE iPreparingToReadyStep OF
	
	0:
		bSwitchOn						:= FALSE;
		bEnableOperation				:= FALSE;						
		bQuickStop						:= FALSE;
		iPreparingToReadyStep			:= 10;	
		
		IF bSwitchedOn THEN
			iPreparingToReadyStep		:= 30;	
		END_IF
		
	10:
		IF bSwitchOnDisabled THEN
		//	bSwitchOn					:= TRUE;
			bEnableVoltage				:= TRUE;						
			bQuickStop					:= TRUE;
			iPreparingToReadyStep		:= 20;	
		END_IF
		
	20:
		IF bReadyToSwitchOn THEN
			bSwitchOn					:= TRUE;
			iPreparingToReadyStep		:= 30;
		END_IF	
	30:
		IF bSwitchedOn THEN
			iPreparingToReadyStep			:= 0;
			eState							:= E_Station.eReady;
			eRunningState					:= E_ConveyorState.eReady;
		END_IF
END_CASE
END_ACTION

ACTION State_Ready:

IF rtRun.Q OR bRun THEN
	bEnableOperation			:= TRUE;
	eState						:= E_Station.eStarting;
	eRunningState				:= E_ConveyorState.eStarting;
END_IF

IF bManualMode THEN
	eState						:= E_Station.eManualMovement;
	eRunningState				:= E_ConveyorState.eManualMovement;
END_IF
END_ACTION

ACTION State_Resetting:

IF bCheckInitTimeError THEN
	bCheckInitTimeError								:= FALSE;
END_IF
IF bWcStateError THEN
	bWcStateError									:= FALSE;
END_IF
IF bMitsubishiReadinessError THEN
	bMitsubishiReadinessError						:= FALSE;
END_IF

IF bExternalError THEN
	bExternalError									:= FALSE;
END_IF
// dodane na testy
IF bFaultReset THEN
	bFaultReset										:=FALSE;
END_IF

IF tonRessetingState.Q THEN
	eState											:= E_Station.eError;
	eRunningState									:= E_ConveyorState.eError;
END_IF

IF NOT bError THEN	
	eState											:= E_Station.ePreparingToReady;	
	eRunningState									:= E_ConveyorState.ePreparingToReady;
END_IF
END_ACTION

ACTION State_Running:


IF NOT bRun THEN
	bEnableOperation					:= FALSE;
	eState								:= E_Station.eStopping;
	eRunningState						:= E_ConveyorState.eStopping;
END_IF
END_ACTION

ACTION State_Starting:
IF bOperationEnabled THEN
	eState							:= E_Station.eRunning;
	eRunningState					:= E_ConveyorState.eWorking;
END_IF

IF NOT bRun THEN
	bEnableOperation				:= FALSE;
	eState							:= E_Station.eStopping;
	eRunningState					:= E_ConveyorState.eStopping;
END_IF
END_ACTION

ACTION State_Stopping:

//bRun dodane na testy
IF NOT bOperationEnabled OR bRun THEN
	eState					:= E_Station.eReady;
	eRunningState			:= E_ConveyorState.eReady;
END_IF
END_ACTION

END_FUNCTION_BLOCK

// ---- POUs/FB/FB_State.TcPOU
(*
Nazwa:			FB_State
Opis:			Generowanie stanów 
Wersja:			v1.0
Data:			2020-04-14
Autor:			DP
Urzadzenia:		
Konfiguracja:	
Info: 
*)

FUNCTION_BLOCK FB_State
VAR_INPUT
	eState							:E_Station;						//Stan ogólny bloku
	bRun							:BOOL;							//Rozkad cyklu	
	eGripperScrewerRunningState		:E_GripperScrewer; 				//Stan zakręcarki szczekowej							
	//eRollerScrewerRunningState		:E_RollerScrewer; 				//Stan zakręcarki rolkowej						
	eCheckerRunningState			:E_CheckerState; 				//Stan sprawdzania
	eEntranceGatesRunningState		:E_EntranceGatesState;			//Stan szlabanów
	eCatchRunningState				:E_CatchStationState;			//Stan wewnętrzny
	eCapPushingRunningState			:E_CapPushingState;				//Stan wbijaka
	eMassHeatingRunningState		:E_MassHeatingState;			//Stan grzania
	eConveyorRunningState			:E_ConveyorState;				//Stan transprterów
	eFormsDragingRunningState 		:E_DragStationState;				//Stan przeciągania zwykłego
	eFormsDragingPneumRunningState	:E_DragStationStatePneum;
	eLidSealingRunningState			:E_LidSealing;					//Stan zgrzewania
	eLidFeederRunningState			:E_LidFeederState;				//Stan platynkowania
	//eWheelRunningState				:E_WheelState;					//Stan kola
	eDispencerRunningState			:E_DispencerState;				//Stan dozowników
	eDispencerLifterRunningState	:E_DispencerLifterState;		//Stan podnośnikow
	eCapFeederRobotRunningState		:E_RobotMovState;				//Stan robota
	eWeightRunningState				:E_WeightState;	
	eWeightLiftRunningState			:E_WeightLiftStationState	;	//Stan wagi		
	eBottleSorterRunningState		:E_BottleFeederState;			// Stan podajnik opakowań		 
	eCapFeederRunningState			:E_CapFeederState;				//Stan podajnika nasadek			
	eWickFeederRunningState			:E_WickFeederState;
END_VAR
VAR_OUTPUT
	sStateDesc						:STRING;
	iState							:INT;							//Stan ogólny bloku
END_VAR
VAR
	iC: INT;
	i: E_DispencerState;
	ic2: INT;
	ic3: INT;
	ic4: INT;
END_VAR


